// SIMATIC STEP 7 (V5.x) project CP#01_OB_PLC(TATA)
// CPU: CPU 315-2 DP
// station: P_ADR_BUS
// station: Hardware
// station: OB_PLC_PC-11
// program: S7 Program(1)

SYMBOL_TABLE
"CMD TO BEC"	DB 10	DB 10	// Command To BEC
"FB FROMBEC"	DB 11	DB 11	// Feedback From BEC
"HMI TAGS"	DB 35	DB 35	// HMI Tags are here
"RDREC"	SFB 52	SFB 52	// Read a Process Data Record
"WRREC"	SFB 53	SFB 53	// Write a Process Data Record
"RD_SINFO"	SFC 6	SFC 6	// Read OB Start Information
"BLKMOV"	SFC 20	SFC 20	// Copy Variables
"FILL"	SFC 21	SFC 21	// Initialize a Memory Area
"RDSYSST"	SFC 51	SFC 51	// Read a System Status List or Partial List
"WR_REC"	SFC 58	SFC 58	// Write Data Record
"RD_REC"	SFC 59	SFC 59	// Read a Data Record
END_SYMBOL_TABLE

// FB 7: know-how protected block, not included

// FB 8: know-how protected block, not included

FUNCTION_BLOCK FB 102
VERSION : 0.0
BEGIN
// body was compiled from an SCL source; compiled code not shown
END_FUNCTION_BLOCK

FUNCTION_BLOCK FB 103
VERSION : 0.0
BEGIN
// body was compiled from an SCL source; compiled code not shown
END_FUNCTION_BLOCK

FUNCTION_BLOCK FB 108
VERSION : 0.0
BEGIN
// body was compiled from an SCL source; compiled code not shown
END_FUNCTION_BLOCK

FUNCTION_BLOCK FB 109
VERSION : 0.0
BEGIN
// body was compiled from an SCL source; compiled code not shown
END_FUNCTION_BLOCK

// FC 1: know-how protected block, not included

// FC 2: know-how protected block, not included

// FC 3: know-how protected block, not included

// FC 4: know-how protected block, not included

FUNCTION FC 10 : VOID
AUTHOR : SKD
NAME : CDSPL
VERSION : 0.1
BEGIN
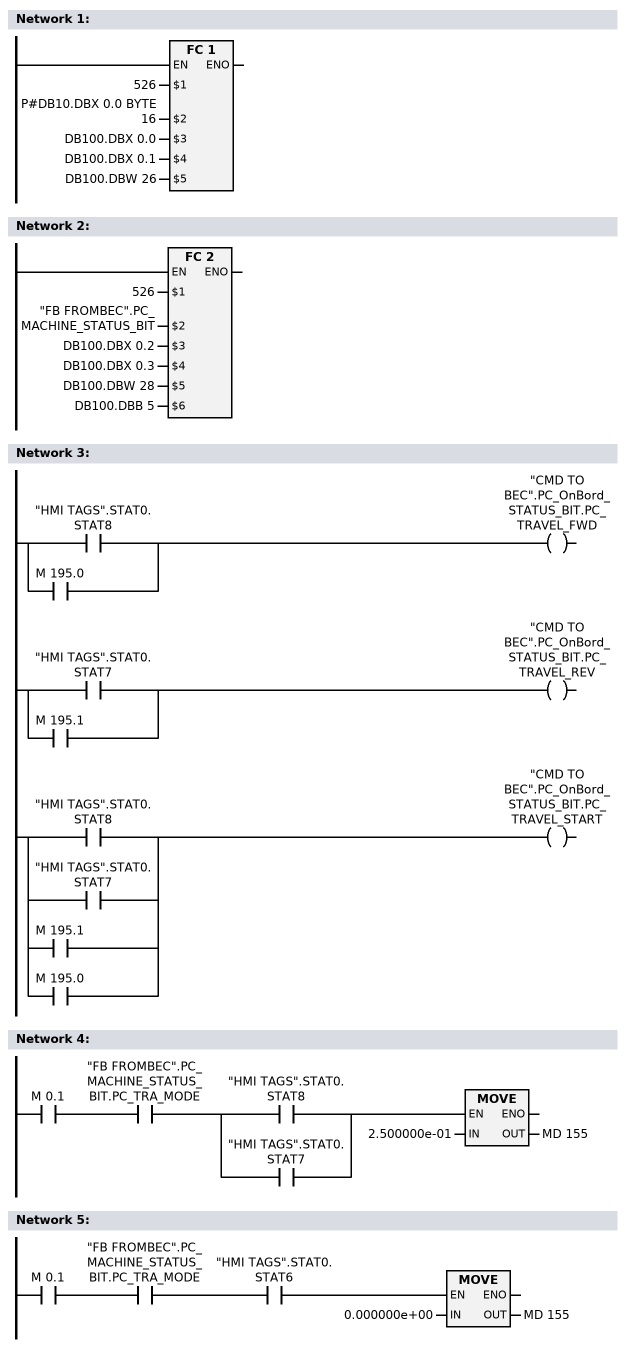
NETWORK
TITLE =
      CALL  FC 1 (
           $1                       := 526,
           $2                       := P#DB10.DBX 0.0 BYTE 16,
           $3                       := DB100.DBX 0.0,
           $4                       := DB100.DBX 0.1,
           $5                       := DB100.DBW 26);
      NOP   0;
NETWORK
TITLE =
      CALL  FC 2 (
           $1                       := 526,
           $2                       := "FB FROMBEC".PC_MACHINE_STATUS_BIT,
           $3                       := DB100.DBX 0.2,
           $4                       := DB100.DBX 0.3,
           $5                       := DB100.DBW 28,
           $6                       := DB100.DBB 5);
      NOP   0;
NETWORK
TITLE =
      O     "HMI TAGS".STAT0.STAT8;
      O     M 195.0;
      =     "CMD TO BEC".PC_OnBord_STATUS_BIT.PC_TRAVEL_FWD;
      O     "HMI TAGS".STAT0.STAT7;
      O     M 195.1;
      =     "CMD TO BEC".PC_OnBord_STATUS_BIT.PC_TRAVEL_REV;
      O     "HMI TAGS".STAT0.STAT8;
      O     "HMI TAGS".STAT0.STAT7;
      O     M 195.1;
      O     M 195.0;
      =     "CMD TO BEC".PC_OnBord_STATUS_BIT.PC_TRAVEL_START;
NETWORK
TITLE =
      A     M 0.1;
      A     "FB FROMBEC".PC_MACHINE_STATUS_BIT.PC_TRA_MODE;
      A(;
      O     "HMI TAGS".STAT0.STAT8;
      O     "HMI TAGS".STAT0.STAT7;
      );
      JNB   _001;
      L     2.500000e-01;
      T     MD 155;
_001: NOP   0;
NETWORK
TITLE =
      A     M 0.1;
      A     "FB FROMBEC".PC_MACHINE_STATUS_BIT.PC_TRA_MODE;
      A     "HMI TAGS".STAT0.STAT6;
      JNB   _002;
      L     0.000000e+00;
      T     MD 155;
_002: NOP   0;
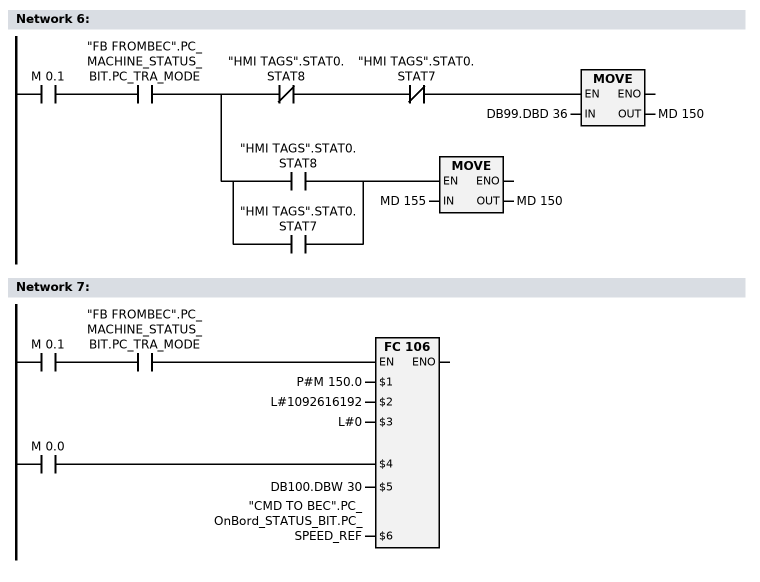
NETWORK
TITLE =
      A     M 0.1;
      A     "FB FROMBEC".PC_MACHINE_STATUS_BIT.PC_TRA_MODE;
      =     L 0.0;
      A     L 0.0;
      AN    "HMI TAGS".STAT0.STAT8;
      AN    "HMI TAGS".STAT0.STAT7;
      JNB   _003;
      L     DB99.DBD 36;
      T     MD 150;
_003: NOP   0;
      A     L 0.0;
      A(;
      O     "HMI TAGS".STAT0.STAT8;
      O     "HMI TAGS".STAT0.STAT7;
      );
      JNB   _004;
      L     MD 155;
      T     MD 150;
_004: NOP   0;
NETWORK
TITLE =
      A     M 0.0;
      =     L 0.0;
      BLD   103;
      A     M 0.1;
      A     "FB FROMBEC".PC_MACHINE_STATUS_BIT.PC_TRA_MODE;
      JNB   _005;
      CALL  FC 106 (
           $1                       := P#M 150.0,
           $2                       := L#1092616192,
           $3                       := L#0,
           $4                       := L 0.0,
           $5                       := DB100.DBW 30,
           $6                       := "CMD TO BEC".PC_OnBord_STATUS_BIT.PC_SPEED_REF);
_005: NOP   0;
END_FUNCTION

FUNCTION FC 14 : VOID
VERSION : 0.1
BEGIN
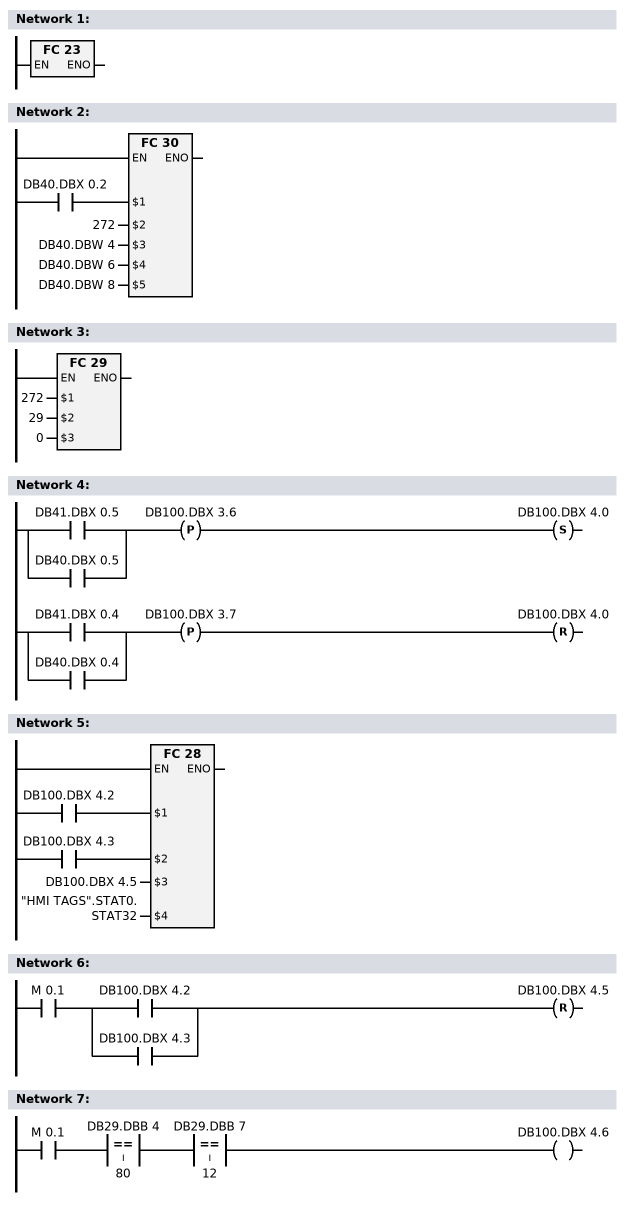
NETWORK
TITLE =
      CALL  FC 23;
      NOP   0;
NETWORK
TITLE =
      A     DB40.DBX 0.2;
      =     L 0.0;
      BLD   103;
      CALL  FC 30 (
           $1                       := L 0.0,
           $2                       := 272,
           $3                       := DB40.DBW 4,
           $4                       := DB40.DBW 6,
           $5                       := DB40.DBW 8);
      NOP   0;
NETWORK
TITLE =
      CALL  FC 29 (
           $1                       := 272,
           $2                       := 29,
           $3                       := 0);
      NOP   0;
NETWORK
TITLE =
      A(;
      O     DB41.DBX 0.5;
      O     DB40.DBX 0.5;
      );
      FP    DB100.DBX 3.6;
      S     DB100.DBX 4.0;
      A(;
      O     DB41.DBX 0.4;
      O     DB40.DBX 0.4;
      );
      FP    DB100.DBX 3.7;
      R     DB100.DBX 4.0;
      NOP   0;
NETWORK
TITLE =
      A     DB100.DBX 4.2;
      =     L 0.0;
      BLD   103;
      A     DB100.DBX 4.3;
      =     L 0.1;
      BLD   103;
      CALL  FC 28 (
           $1                       := L 0.0,
           $2                       := L 0.1,
           $3                       := DB100.DBX 4.5,
           $4                       := "HMI TAGS".STAT0.STAT32);
      NOP   0;
NETWORK
TITLE =
      A     M 0.1;
      A(;
      O     DB100.DBX 4.2;
      O     DB100.DBX 4.3;
      );
      R     DB100.DBX 4.5;
NETWORK
TITLE =
      A     M 0.1;
      A(;
      L     DB29.DBB 4;
      L     80;
      ==I;
      );
      A(;
      L     DB29.DBB 7;
      L     12;
      ==I;
      );
      =     DB100.DBX 4.6;
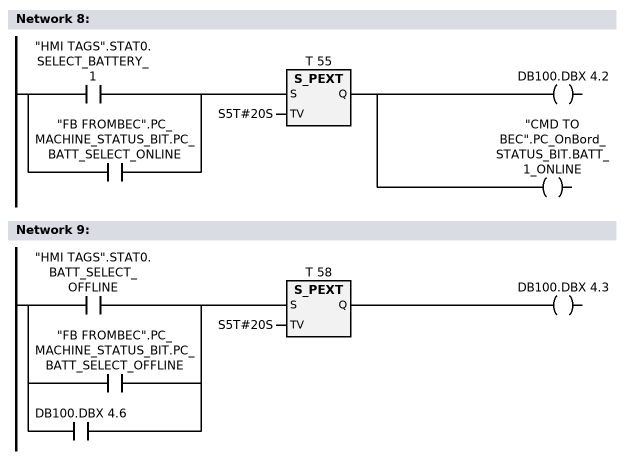
NETWORK
TITLE =
      A(;
      O     "HMI TAGS".STAT0.SELECT_BATTERY_1;
      O     "FB FROMBEC".PC_MACHINE_STATUS_BIT.PC_BATT_SELECT_ONLINE;
      );
      L     S5T#20S;
      SE    T 55;
      NOP   0;
      NOP   0;
      NOP   0;
      A     T 55;
      =     DB100.DBX 4.2;
      =     "CMD TO BEC".PC_OnBord_STATUS_BIT.BATT_1_ONLINE;
NETWORK
TITLE =
      A(;
      O     "HMI TAGS".STAT0.BATT_SELECT_OFFLINE;
      O     "FB FROMBEC".PC_MACHINE_STATUS_BIT.PC_BATT_SELECT_OFFLINE;
      O     DB100.DBX 4.6;
      );
      L     S5T#20S;
      SE    T 58;
      NOP   0;
      NOP   0;
      NOP   0;
      A     T 58;
      =     DB100.DBX 4.3;
END_FUNCTION

FUNCTION FC 16 : VOID
VERSION : 0.1
BEGIN
// (block stored without names or comments; labels and parameter names are numbered)
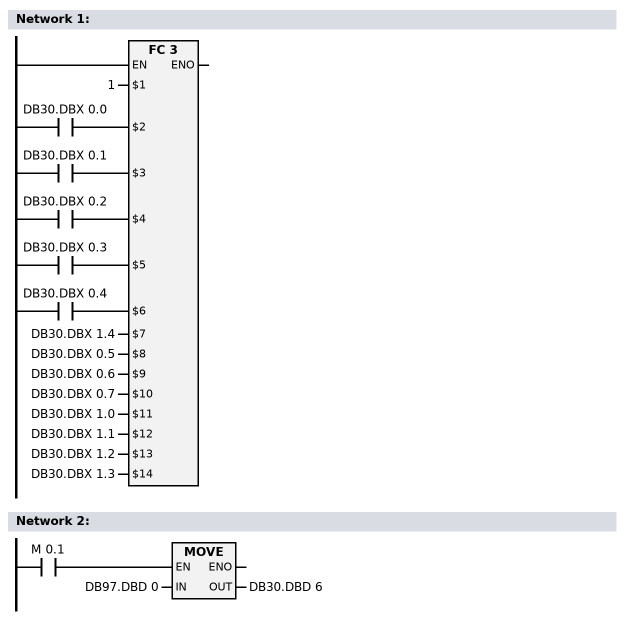
NETWORK
TITLE =
      A     DB30.DBX 0.0;
      =     L 4.0;
      BLD   103;
      A     DB30.DBX 0.1;
      =     L 4.1;
      BLD   103;
      A     DB30.DBX 0.2;
      =     L 4.2;
      BLD   103;
      A     DB30.DBX 0.3;
      =     L 4.3;
      BLD   103;
      A     DB30.DBX 0.4;
      =     L 4.4;
      BLD   103;
      CALL  FC 3 (
           $1                       := 1,
           $2                       := L 4.0,
           $3                       := L 4.1,
           $4                       := L 4.2,
           $5                       := L 4.3,
           $6                       := L 4.4,
           $7                       := DB30.DBX 1.4,
           $8                       := DB30.DBX 0.5,
           $9                       := DB30.DBX 0.6,
           $10                      := DB30.DBX 0.7,
           $11                      := DB30.DBX 1.0,
           $12                      := DB30.DBX 1.1,
           $13                      := DB30.DBX 1.2,
           $14                      := DB30.DBX 1.3);
      NOP   0;
NETWORK
TITLE =
      A     M 0.1;
      JNB   M001;
      L     DB97.DBD 0;
      T     DB30.DBD 6;
M001: NOP   0;
END_FUNCTION

FUNCTION FC 19 : VOID
VERSION : 0.1
BEGIN
// (block stored without names or comments; labels and parameter names are numbered)
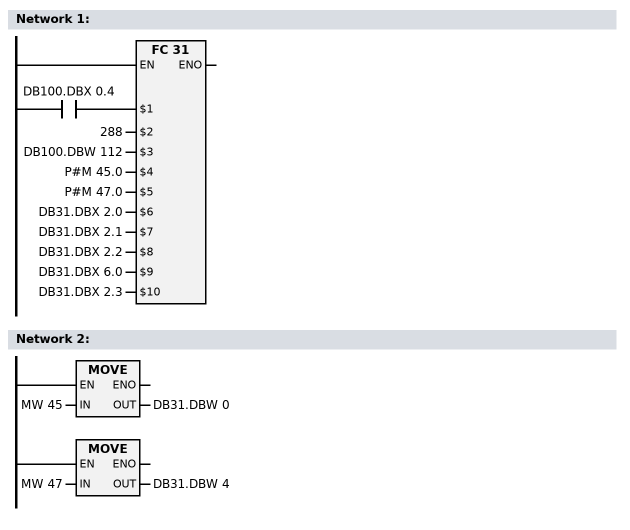
NETWORK
TITLE =
      A     DB100.DBX 0.4;
      =     L 0.0;
      BLD   103;
      CALL  FC 31 (
           $1                       := L 0.0,
           $2                       := 288,
           $3                       := DB100.DBW 112,
           $4                       := P#M 45.0,
           $5                       := P#M 47.0,
           $6                       := DB31.DBX 2.0,
           $7                       := DB31.DBX 2.1,
           $8                       := DB31.DBX 2.2,
           $9                       := DB31.DBX 6.0,
           $10                      := DB31.DBX 2.3);
      NOP   0;
NETWORK
TITLE =
      L     MW 45;
      T     DB31.DBW 0;
      L     MW 47;
      T     DB31.DBW 4;
END_FUNCTION

FUNCTION FC 20 : VOID
VERSION : 0.1
BEGIN
// (block stored without names or comments; labels and parameter names are numbered)
NETWORK
TITLE =
      A     M 0.1;
      A(;
      L     DB21.DBW 46;
      L     1;
      ==I;
      );
      A(;
      L     DB21.DBB 50;
      L     'P';
      ==I;
      );
      JNB   M001;
      L     DB21.DBW 24;
      T     "HMI TAGS".STAT98.STAT120;
M001: NOP   0;
NETWORK
TITLE =
      A     M 0.1;
      A(;
      L     DB21.DBW 46;
      L     1;
      ==I;
      );
      A(;
      L     DB21.DBB 50;
      L     'C';
      ==I;
      );
      A(;
      L     DB21.DBW 74;
      L     2;
      ==I;
      );
      A(;
      L     DB21.DBB 78;
      L     'P';
      ==I;
      );
      JNB   M002;
      L     DB21.DBW 52;
      T     "HMI TAGS".STAT98.STAT120;
M002: NOP   0;
NETWORK
TITLE =
      A     M 0.1;
      A(;
      L     DB21.DBW 46;
      L     1;
      ==I;
      );
      A(;
      L     DB21.DBB 50;
      L     'C';
      ==I;
      );
      A(;
      L     DB21.DBW 74;
      L     2;
      ==I;
      );
      A(;
      L     DB21.DBB 78;
      L     'C';
      ==I;
      );
      A(;
      L     DB21.DBW 102;
      L     3;
      ==I;
      );
      A(;
      L     DB21.DBB 106;
      L     'P';
      ==I;
      );
      JNB   M003;
      L     DB21.DBW 80;
      T     "HMI TAGS".STAT98.STAT120;
M003: NOP   0;
NETWORK
TITLE =
      A     M 0.1;
      A(;
      L     DB21.DBW 46;
      L     1;
      ==I;
      );
      A(;
      L     DB21.DBB 50;
      L     'C';
      ==I;
      );
      A(;
      L     DB21.DBW 74;
      L     2;
      ==I;
      );
      A(;
      L     DB21.DBB 78;
      L     'C';
      ==I;
      );
      A(;
      L     DB21.DBW 102;
      L     3;
      ==I;
      );
      A(;
      L     DB21.DBB 106;
      L     'C';
      ==I;
      );
      A(;
      L     DB21.DBW 130;
      L     4;
      ==I;
      );
      A(;
      L     DB21.DBB 134;
      L     'P';
      ==I;
      );
      JNB   M004;
      L     DB21.DBW 108;
      T     "HMI TAGS".STAT98.STAT120;
M004: NOP   0;
NETWORK
TITLE =
      A     M 0.1;
      A(;
      L     DB21.DBW 46;
      L     1;
      ==I;
      );
      A(;
      L     DB21.DBB 50;
      L     'C';
      ==I;
      );
      =     L 0.0;
      A     L 0.0;
      JNB   M005;
      L     DB21.DBW 24;
      T     "HMI TAGS".STAT98.STAT121;
M005: NOP   0;
      A     L 0.0;
      JNB   M006;
      L     DB21.DBB 50;
      T     DB35.DBB 284;
M006: NOP   0;
END_FUNCTION

FUNCTION FC 21 : VOID
VERSION : 0.1
BEGIN
// (block stored without names or comments; labels and parameter names are numbered)
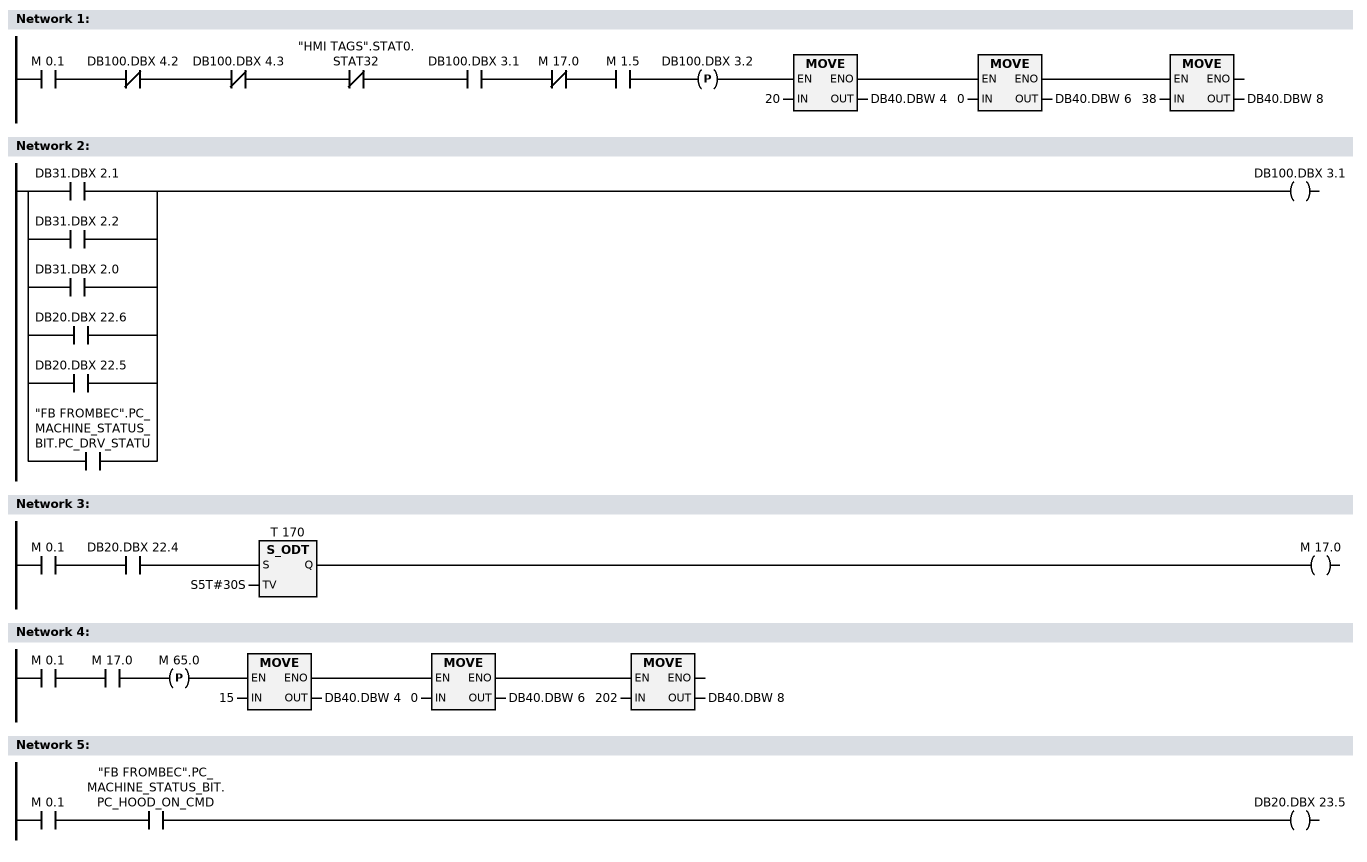
NETWORK
TITLE =
      A(;
      A(;
      A     M 0.1;
      AN    DB100.DBX 4.2;
      AN    DB100.DBX 4.3;
      AN    "HMI TAGS".STAT0.STAT32;
      A     DB100.DBX 3.1;
      AN    M 17.0;
      A     M 1.5;
      FP    DB100.DBX 3.2;
      JNB   M001;
      L     20;
      T     DB40.DBW 4;
      SET;
      SAVE;
      CLR;
M001: A     BR;
      );
      JNB   M002;
      L     0;
      T     DB40.DBW 6;
      SET;
      SAVE;
      CLR;
M002: A     BR;
      );
      JNB   M003;
      L     38;
      T     DB40.DBW 8;
M003: NOP   0;
NETWORK
TITLE =
      O     DB31.DBX 2.1;
      O     DB31.DBX 2.2;
      O     DB31.DBX 2.0;
      O     DB20.DBX 22.6;
      O     DB20.DBX 22.5;
      O     "FB FROMBEC".PC_MACHINE_STATUS_BIT.PC_DRV_STATU;
      =     DB100.DBX 3.1;
NETWORK
TITLE =
      A     M 0.1;
      A     DB20.DBX 22.4;
      L     S5T#30S;
      SD    T 170;
      NOP   0;
      NOP   0;
      NOP   0;
      A     T 170;
      =     M 17.0;
NETWORK
TITLE =
      A(;
      A(;
      A     M 0.1;
      A     M 17.0;
      FP    M 65.0;
      JNB   M004;
      L     15;
      T     DB40.DBW 4;
      SET;
      SAVE;
      CLR;
M004: A     BR;
      );
      JNB   M005;
      L     0;
      T     DB40.DBW 6;
      SET;
      SAVE;
      CLR;
M005: A     BR;
      );
      JNB   M006;
      L     202;
      T     DB40.DBW 8;
M006: NOP   0;
NETWORK
TITLE =
      A     M 0.1;
      A     "FB FROMBEC".PC_MACHINE_STATUS_BIT.PC_HOOD_ON_CMD;
      =     DB20.DBX 23.5;
NETWORK
TITLE =
      BE;
END_FUNCTION

FUNCTION FC 22 : VOID
VERSION : 0.1
BEGIN
// (block stored without names or comments; labels and parameter names are numbered)
NETWORK
TITLE =
      A     DB41.DBX 0.4;
      A(;
      L     DB29.DBB 8;
      L     B#16#3;
      ==I;
      );
      A(;
      L     DB29.DBB 11;
      L     32;
      ==I;
      );
      =     DB100.DBX 15.1;
      A     DB100.DBX 15.1;
      JNB   M001;
      CALL  "FILL" (
           BVAL                     := P#DB29.DBX 0.0 BYTE 30,
           RET_VAL                  := DB100.DBW 122,
           BLK                      := P#DB17.DBX 0.0 BYTE 30);
M001: NOP   0;
NETWORK
TITLE =
      A     DB41.DBX 0.4;
      A(;
      L     DB29.DBB 8;
      L     B#16#4;
      ==I;
      );
      A(;
      L     DB29.DBB 11;
      L     30;
      ==I;
      );
      =     DB100.DBX 15.2;
      A     DB100.DBX 15.2;
      JNB   M002;
      CALL  "FILL" (
           BVAL                     := P#DB29.DBX 0.0 BYTE 30,
           RET_VAL                  := DB100.DBW 124,
           BLK                      := P#DB19.DBX 0.0 BYTE 30);
M002: NOP   0;
NETWORK
TITLE =
      A     DB41.DBX 0.4;
      A(;
      L     DB29.DBB 8;
      L     B#16#5;
      ==I;
      );
      A(;
      L     DB29.DBB 11;
      L     34;
      ==I;
      );
      =     DB100.DBX 15.3;
      A     DB100.DBX 15.3;
      FP    DB100.DBX 15.5;
      JNB   M003;
      CALL  "FILL" (
           BVAL                     := P#DB29.DBX 0.0 BYTE 34,
           RET_VAL                  := DB100.DBW 126,
           BLK                      := P#DB18.DBX 0.0 BYTE 34);
M003: NOP   0;
NETWORK
TITLE =
      A     DB41.DBX 0.4;
      A(;
      L     DB29.DBB 8;
      L     B#16#10;
      ==I;
      );
      A(;
      L     DB29.DBB 11;
      L     167;
      ==I;
      );
      =     DB100.DBX 15.4;
      A     DB100.DBX 15.4;
      JNB   M004;
      CALL  "FILL" (
           BVAL                     := P#DB29.DBX 0.0 BYTE 167,
           RET_VAL                  := DB100.DBW 128,
           BLK                      := P#DB21.DBX 0.0 BYTE 167);
M004: NOP   0;
END_FUNCTION

FUNCTION FC 23 : VOID
VERSION : 0.1
BEGIN
// (block stored without names or comments; labels and parameter names are numbered)
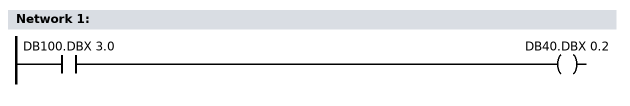
NETWORK
TITLE =
      A     DB100.DBX 3.0;
      =     DB40.DBX 0.2;
END_FUNCTION

FUNCTION FC 24 : VOID
VERSION : 0.1
BEGIN
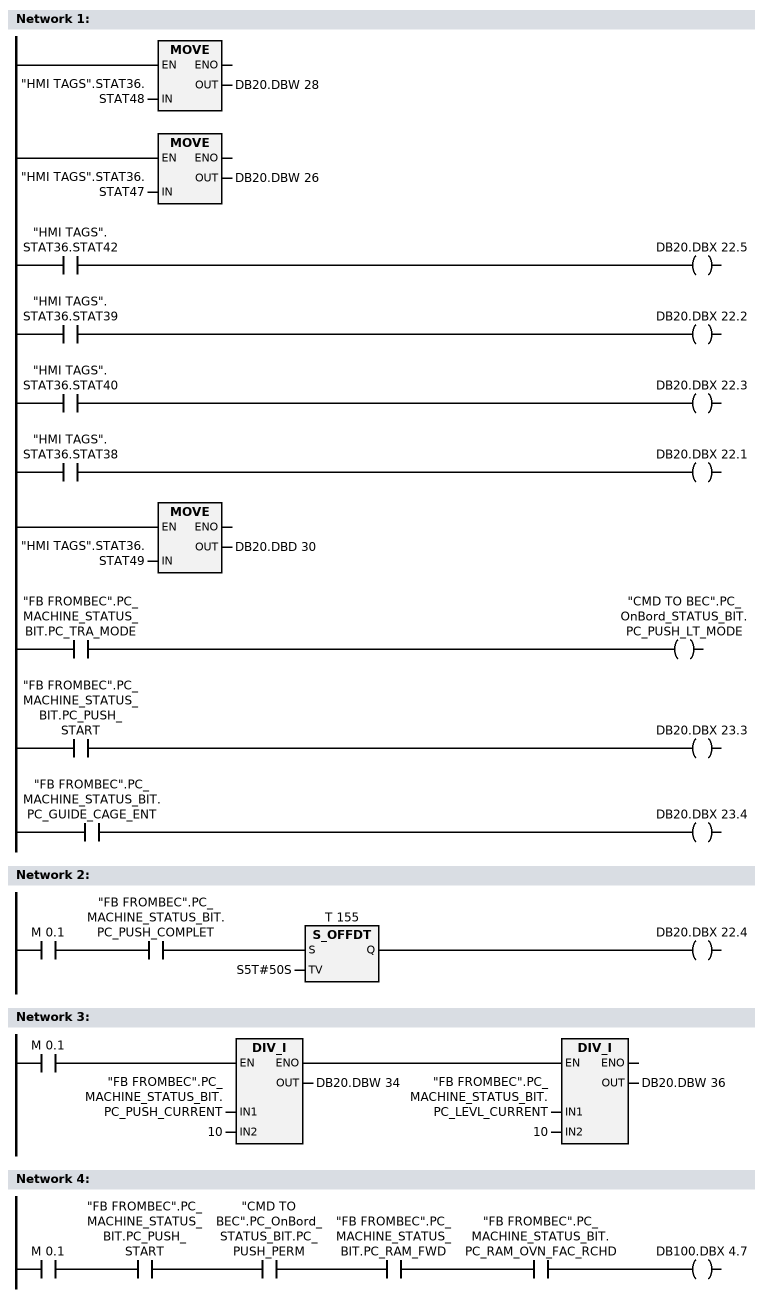
NETWORK
TITLE =
      L     "HMI TAGS".STAT36.STAT48;
      T     DB20.DBW 28;
      L     "HMI TAGS".STAT36.STAT47;
      T     DB20.DBW 26;
      A     "HMI TAGS".STAT36.STAT42;
      =     DB20.DBX 22.5;
      A     "HMI TAGS".STAT36.STAT39;
      =     DB20.DBX 22.2;
      A     "HMI TAGS".STAT36.STAT40;
      =     DB20.DBX 22.3;
      A     "HMI TAGS".STAT36.STAT38;
      =     DB20.DBX 22.1;
      L     "HMI TAGS".STAT36.STAT49;
      T     DB20.DBD 30;
      A     "FB FROMBEC".PC_MACHINE_STATUS_BIT.PC_TRA_MODE;
      =     "CMD TO BEC".PC_OnBord_STATUS_BIT.PC_PUSH_LT_MODE;
      A     "FB FROMBEC".PC_MACHINE_STATUS_BIT.PC_PUSH_START;
      =     DB20.DBX 23.3;
      A     "FB FROMBEC".PC_MACHINE_STATUS_BIT.PC_GUIDE_CAGE_ENT;
      =     DB20.DBX 23.4;
NETWORK
TITLE =
      A     M 0.1;
      A     "FB FROMBEC".PC_MACHINE_STATUS_BIT.PC_PUSH_COMPLET;
      L     S5T#50S;
      SF    T 155;
      NOP   0;
      NOP   0;
      NOP   0;
      A     T 155;
      =     DB20.DBX 22.4;
NETWORK
TITLE =
      A(;
      A     M 0.1;
      JNB   _001;
      L     "FB FROMBEC".PC_MACHINE_STATUS_BIT.PC_PUSH_CURRENT;
      L     10;
      /I;
      T     DB20.DBW 34;
      AN    OV;
      SAVE;
      CLR;
_001: A     BR;
      );
      JNB   _002;
      L     "FB FROMBEC".PC_MACHINE_STATUS_BIT.PC_LEVL_CURRENT;
      L     10;
      /I;
      T     DB20.DBW 36;
_002: NOP   0;
NETWORK
TITLE =
      A     M 0.1;
      A     "FB FROMBEC".PC_MACHINE_STATUS_BIT.PC_PUSH_START;
      A     "CMD TO BEC".PC_OnBord_STATUS_BIT.PC_PUSH_PERM;
      A     "FB FROMBEC".PC_MACHINE_STATUS_BIT.PC_RAM_FWD;
      A     "FB FROMBEC".PC_MACHINE_STATUS_BIT.PC_RAM_OVN_FAC_RCHD;
      =     DB100.DBX 4.7;
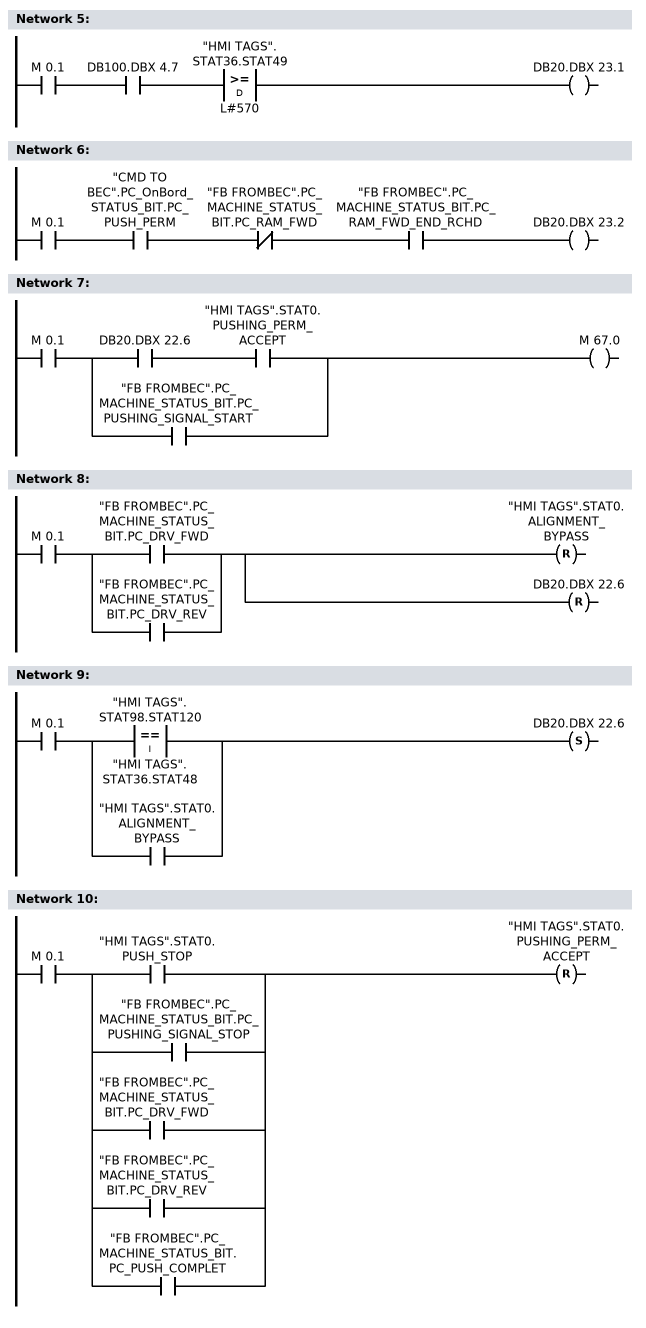
NETWORK
TITLE =
      A     M 0.1;
      A     DB100.DBX 4.7;
      A(;
      L     "HMI TAGS".STAT36.STAT49;
      L     L#570;
      >=D;
      );
      =     DB20.DBX 23.1;
NETWORK
TITLE =
      A     M 0.1;
      A     "CMD TO BEC".PC_OnBord_STATUS_BIT.PC_PUSH_PERM;
      AN    "FB FROMBEC".PC_MACHINE_STATUS_BIT.PC_RAM_FWD;
      A     "FB FROMBEC".PC_MACHINE_STATUS_BIT.PC_RAM_FWD_END_RCHD;
      =     DB20.DBX 23.2;
NETWORK
TITLE =
      A     M 0.1;
      A(;
      A     DB20.DBX 22.6;
      A     "HMI TAGS".STAT0.PUSHING_PERM_ACCEPT;
      O     "FB FROMBEC".PC_MACHINE_STATUS_BIT.PC_PUSHING_SIGNAL_START;
      );
      =     M 67.0;
NETWORK
TITLE =
      A     M 0.1;
      A(;
      O     "FB FROMBEC".PC_MACHINE_STATUS_BIT.PC_DRV_FWD;
      O     "FB FROMBEC".PC_MACHINE_STATUS_BIT.PC_DRV_REV;
      );
      R     "HMI TAGS".STAT0.ALIGNMENT_BYPASS;
      R     DB20.DBX 22.6;
NETWORK
TITLE =
      A     M 0.1;
      A(;
      O(;
      L     "HMI TAGS".STAT98.STAT120;
      L     "HMI TAGS".STAT36.STAT48;
      ==I;
      );
      O     "HMI TAGS".STAT0.ALIGNMENT_BYPASS;
      );
      S     DB20.DBX 22.6;
NETWORK
TITLE =
      A     M 0.1;
      A(;
      O     "HMI TAGS".STAT0.PUSH_STOP;
      O     "FB FROMBEC".PC_MACHINE_STATUS_BIT.PC_PUSHING_SIGNAL_STOP;
      O     "FB FROMBEC".PC_MACHINE_STATUS_BIT.PC_DRV_FWD;
      O     "FB FROMBEC".PC_MACHINE_STATUS_BIT.PC_DRV_REV;
      O     "FB FROMBEC".PC_MACHINE_STATUS_BIT.PC_PUSH_COMPLET;
      );
      R     "HMI TAGS".STAT0.PUSHING_PERM_ACCEPT;
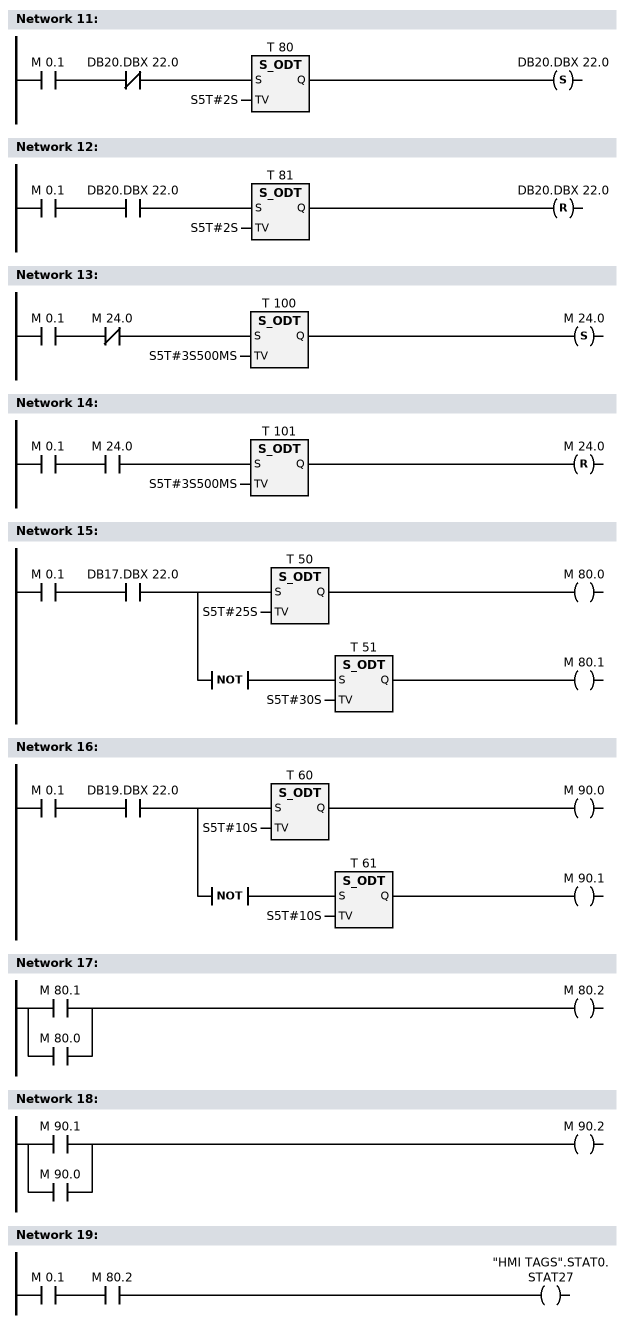
NETWORK
TITLE =
      A     M 0.1;
      AN    DB20.DBX 22.0;
      L     S5T#2S;
      SD    T 80;
      NOP   0;
      NOP   0;
      NOP   0;
      A     T 80;
      S     DB20.DBX 22.0;
NETWORK
TITLE =
      A     M 0.1;
      A     DB20.DBX 22.0;
      L     S5T#2S;
      SD    T 81;
      NOP   0;
      NOP   0;
      NOP   0;
      A     T 81;
      R     DB20.DBX 22.0;
NETWORK
TITLE =
      A     M 0.1;
      AN    M 24.0;
      L     S5T#3S500MS;
      SD    T 100;
      NOP   0;
      NOP   0;
      NOP   0;
      A     T 100;
      S     M 24.0;
NETWORK
TITLE =
      A     M 0.1;
      A     M 24.0;
      L     S5T#3S500MS;
      SD    T 101;
      NOP   0;
      NOP   0;
      NOP   0;
      A     T 101;
      R     M 24.0;
NETWORK
TITLE =
      A     M 0.1;
      A     DB17.DBX 22.0;
      =     L 0.0;
      A     L 0.0;
      L     S5T#25S;
      SD    T 50;
      NOP   0;
      NOP   0;
      NOP   0;
      A     T 50;
      =     M 80.0;
      A     L 0.0;
      NOT;
      L     S5T#30S;
      SD    T 51;
      NOP   0;
      NOP   0;
      NOP   0;
      A     T 51;
      =     M 80.1;
NETWORK
TITLE =
      A     M 0.1;
      A     DB19.DBX 22.0;
      =     L 0.0;
      A     L 0.0;
      L     S5T#10S;
      SD    T 60;
      NOP   0;
      NOP   0;
      NOP   0;
      A     T 60;
      =     M 90.0;
      A     L 0.0;
      NOT;
      L     S5T#10S;
      SD    T 61;
      NOP   0;
      NOP   0;
      NOP   0;
      A     T 61;
      =     M 90.1;
NETWORK
TITLE =
      O     M 80.1;
      O     M 80.0;
      =     M 80.2;
NETWORK
TITLE =
      O     M 90.1;
      O     M 90.0;
      =     M 90.2;
NETWORK
TITLE =
      A     M 0.1;
      A     M 80.2;
      =     "HMI TAGS".STAT0.STAT27;
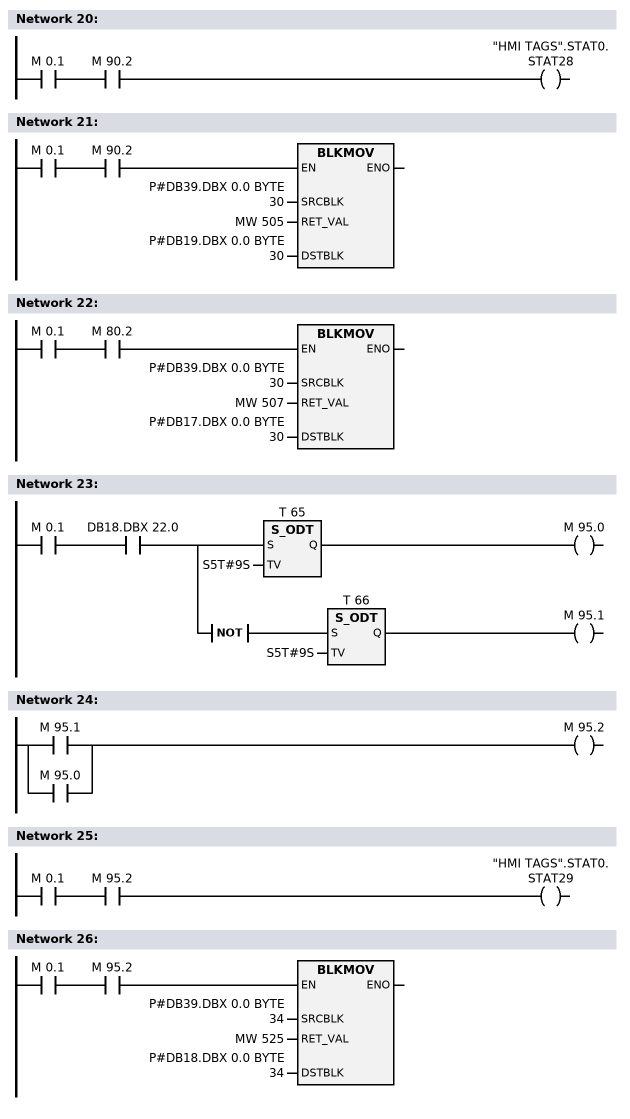
NETWORK
TITLE =
      A     M 0.1;
      A     M 90.2;
      =     "HMI TAGS".STAT0.STAT28;
NETWORK
TITLE =
      A     M 0.1;
      A     M 90.2;
      JNB   _003;
      CALL  "BLKMOV" (
           SRCBLK                   := P#DB39.DBX 0.0 BYTE 30,
           RET_VAL                  := MW 505,
           DSTBLK                   := P#DB19.DBX 0.0 BYTE 30);
_003: NOP   0;
NETWORK
TITLE =
      A     M 0.1;
      A     M 80.2;
      JNB   _004;
      CALL  "BLKMOV" (
           SRCBLK                   := P#DB39.DBX 0.0 BYTE 30,
           RET_VAL                  := MW 507,
           DSTBLK                   := P#DB17.DBX 0.0 BYTE 30);
_004: NOP   0;
NETWORK
TITLE =
      A     M 0.1;
      A     DB18.DBX 22.0;
      =     L 0.0;
      A     L 0.0;
      L     S5T#9S;
      SD    T 65;
      NOP   0;
      NOP   0;
      NOP   0;
      A     T 65;
      =     M 95.0;
      A     L 0.0;
      NOT;
      L     S5T#9S;
      SD    T 66;
      NOP   0;
      NOP   0;
      NOP   0;
      A     T 66;
      =     M 95.1;
NETWORK
TITLE =
      O     M 95.1;
      O     M 95.0;
      =     M 95.2;
NETWORK
TITLE =
      A     M 0.1;
      A     M 95.2;
      =     "HMI TAGS".STAT0.STAT29;
NETWORK
TITLE =
      A     M 0.1;
      A     M 95.2;
      JNB   _005;
      CALL  "BLKMOV" (
           SRCBLK                   := P#DB39.DBX 0.0 BYTE 34,
           RET_VAL                  := MW 525,
           DSTBLK                   := P#DB18.DBX 0.0 BYTE 34);
_005: NOP   0;
END_FUNCTION

FUNCTION FC 26 : VOID
VERSION : 0.1
BEGIN
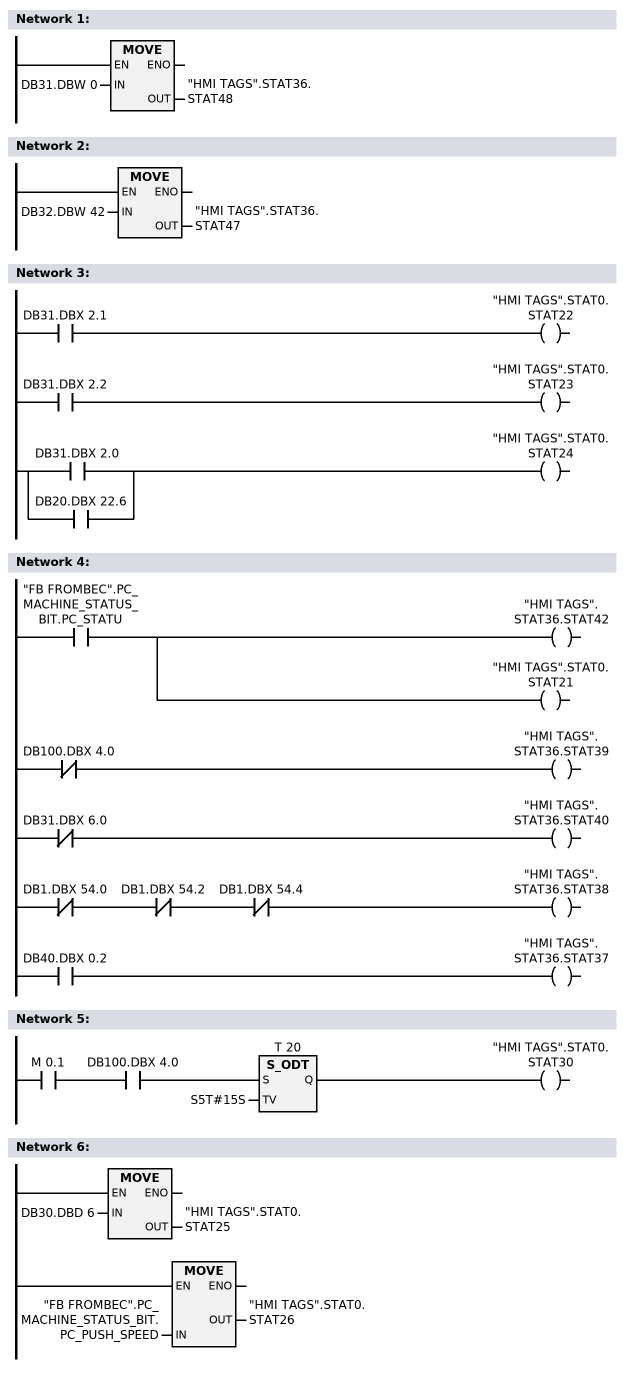
NETWORK
TITLE =
      L     DB31.DBW 0;
      T     "HMI TAGS".STAT36.STAT48;
NETWORK
TITLE =
      L     DB32.DBW 42;
      T     "HMI TAGS".STAT36.STAT47;
NETWORK
TITLE =
      A     DB31.DBX 2.1;
      =     "HMI TAGS".STAT0.STAT22;
      A     DB31.DBX 2.2;
      =     "HMI TAGS".STAT0.STAT23;
      O     DB31.DBX 2.0;
      O     DB20.DBX 22.6;
      =     "HMI TAGS".STAT0.STAT24;
NETWORK
TITLE =
      A     "FB FROMBEC".PC_MACHINE_STATUS_BIT.PC_STATU;
      =     "HMI TAGS".STAT36.STAT42;
      =     "HMI TAGS".STAT0.STAT21;
      AN    DB100.DBX 4.0;
      =     "HMI TAGS".STAT36.STAT39;
      AN    DB31.DBX 6.0;
      =     "HMI TAGS".STAT36.STAT40;
      AN    DB1.DBX 54.0;
      AN    DB1.DBX 54.2;
      AN    DB1.DBX 54.4;
      =     "HMI TAGS".STAT36.STAT38;
      A     DB40.DBX 0.2;
      =     "HMI TAGS".STAT36.STAT37;
NETWORK
TITLE =
      A     M 0.1;
      A     DB100.DBX 4.0;
      L     S5T#15S;
      SD    T 20;
      NOP   0;
      NOP   0;
      NOP   0;
      A     T 20;
      =     "HMI TAGS".STAT0.STAT30;
NETWORK
TITLE =
      L     DB30.DBD 6;
      T     "HMI TAGS".STAT0.STAT25;
      L     "FB FROMBEC".PC_MACHINE_STATUS_BIT.PC_PUSH_SPEED;
      T     "HMI TAGS".STAT0.STAT26;
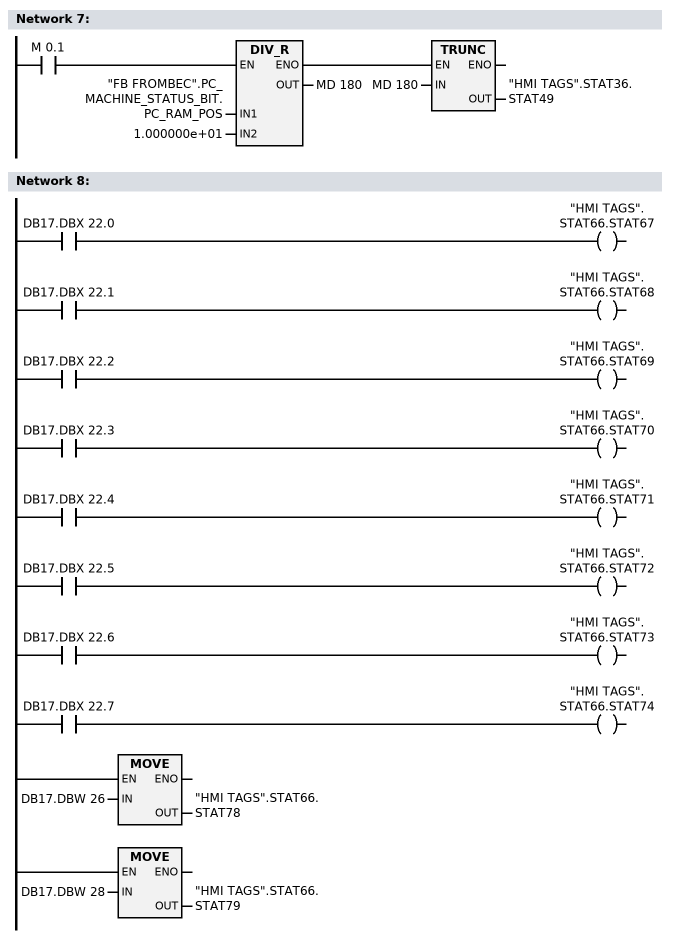
NETWORK
TITLE =
      A(;
      A     M 0.1;
      JNB   _001;
      L     "FB FROMBEC".PC_MACHINE_STATUS_BIT.PC_RAM_POS;
      L     1.000000e+01;
      /R;
      T     MD 180;
      AN    OV;
      SAVE;
      CLR;
_001: A     BR;
      );
      JNB   _002;
      L     MD 180;
      TRUNC;
      T     "HMI TAGS".STAT36.STAT49;
_002: NOP   0;
NETWORK
TITLE =
      A     DB17.DBX 22.0;
      =     "HMI TAGS".STAT66.STAT67;
      A     DB17.DBX 22.1;
      =     "HMI TAGS".STAT66.STAT68;
      A     DB17.DBX 22.2;
      =     "HMI TAGS".STAT66.STAT69;
      A     DB17.DBX 22.3;
      =     "HMI TAGS".STAT66.STAT70;
      A     DB17.DBX 22.4;
      =     "HMI TAGS".STAT66.STAT71;
      A     DB17.DBX 22.5;
      =     "HMI TAGS".STAT66.STAT72;
      A     DB17.DBX 22.6;
      =     "HMI TAGS".STAT66.STAT73;
      A     DB17.DBX 22.7;
      =     "HMI TAGS".STAT66.STAT74;
      L     DB17.DBW 26;
      T     "HMI TAGS".STAT66.STAT78;
      L     DB17.DBW 28;
      T     "HMI TAGS".STAT66.STAT79;
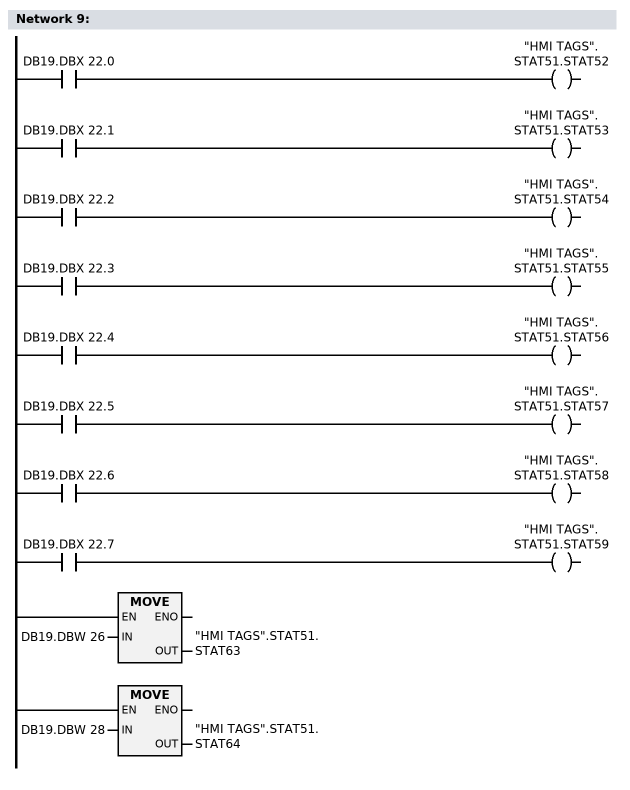
NETWORK
TITLE =
      A     DB19.DBX 22.0;
      =     "HMI TAGS".STAT51.STAT52;
      A     DB19.DBX 22.1;
      =     "HMI TAGS".STAT51.STAT53;
      A     DB19.DBX 22.2;
      =     "HMI TAGS".STAT51.STAT54;
      A     DB19.DBX 22.3;
      =     "HMI TAGS".STAT51.STAT55;
      A     DB19.DBX 22.4;
      =     "HMI TAGS".STAT51.STAT56;
      A     DB19.DBX 22.5;
      =     "HMI TAGS".STAT51.STAT57;
      A     DB19.DBX 22.6;
      =     "HMI TAGS".STAT51.STAT58;
      A     DB19.DBX 22.7;
      =     "HMI TAGS".STAT51.STAT59;
      L     DB19.DBW 26;
      T     "HMI TAGS".STAT51.STAT63;
      L     DB19.DBW 28;
      T     "HMI TAGS".STAT51.STAT64;
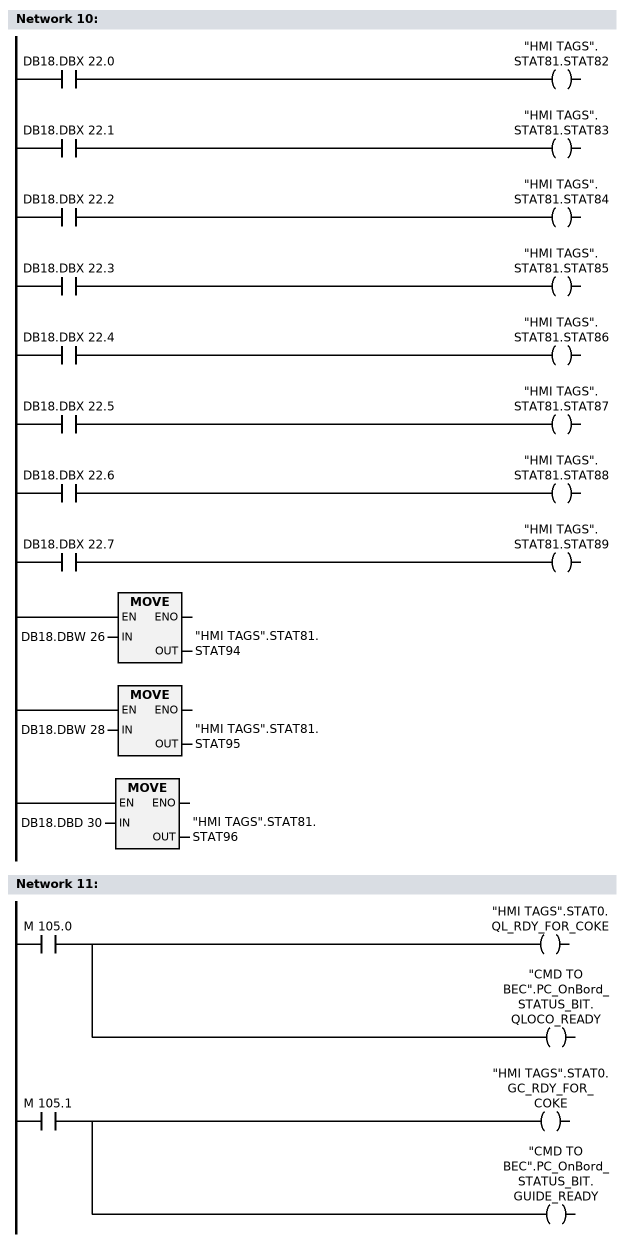
NETWORK
TITLE =
      A     DB18.DBX 22.0;
      =     "HMI TAGS".STAT81.STAT82;
      A     DB18.DBX 22.1;
      =     "HMI TAGS".STAT81.STAT83;
      A     DB18.DBX 22.2;
      =     "HMI TAGS".STAT81.STAT84;
      A     DB18.DBX 22.3;
      =     "HMI TAGS".STAT81.STAT85;
      A     DB18.DBX 22.4;
      =     "HMI TAGS".STAT81.STAT86;
      A     DB18.DBX 22.5;
      =     "HMI TAGS".STAT81.STAT87;
      A     DB18.DBX 22.6;
      =     "HMI TAGS".STAT81.STAT88;
      A     DB18.DBX 22.7;
      =     "HMI TAGS".STAT81.STAT89;
      L     DB18.DBW 26;
      T     "HMI TAGS".STAT81.STAT94;
      L     DB18.DBW 28;
      T     "HMI TAGS".STAT81.STAT95;
      L     DB18.DBD 30;
      T     "HMI TAGS".STAT81.STAT96;
NETWORK
TITLE =
      A     M 105.0;
      =     "HMI TAGS".STAT0.QL_RDY_FOR_COKE;
      =     "CMD TO BEC".PC_OnBord_STATUS_BIT.QLOCO_READY;
      A     M 105.1;
      =     "HMI TAGS".STAT0.GC_RDY_FOR_COKE;
      =     "CMD TO BEC".PC_OnBord_STATUS_BIT.GUIDE_READY;
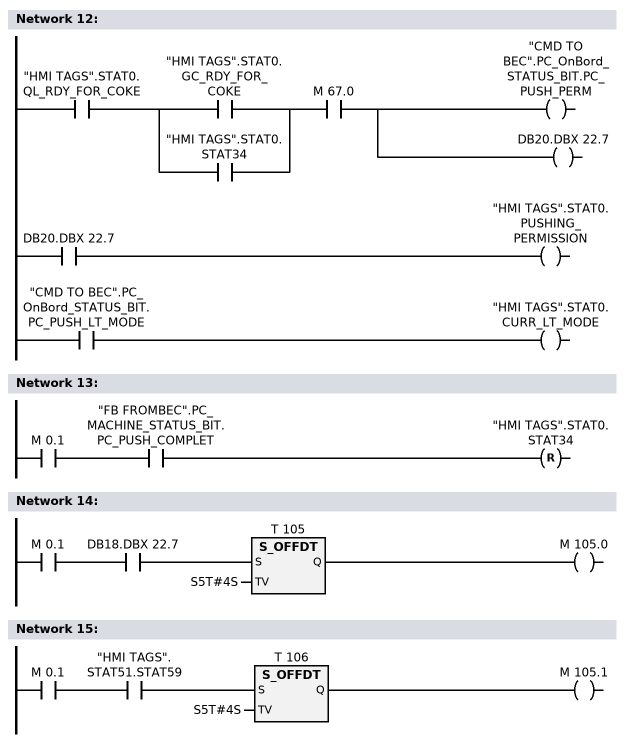
NETWORK
TITLE =
      A     "HMI TAGS".STAT0.QL_RDY_FOR_COKE;
      A(;
      O     "HMI TAGS".STAT0.GC_RDY_FOR_COKE;
      O     "HMI TAGS".STAT0.STAT34;
      );
      A     M 67.0;
      =     "CMD TO BEC".PC_OnBord_STATUS_BIT.PC_PUSH_PERM;
      =     DB20.DBX 22.7;
      A     DB20.DBX 22.7;
      =     "HMI TAGS".STAT0.PUSHING_PERMISSION;
      A     "CMD TO BEC".PC_OnBord_STATUS_BIT.PC_PUSH_LT_MODE;
      =     "HMI TAGS".STAT0.CURR_LT_MODE;
NETWORK
TITLE =
      A     M 0.1;
      A     "FB FROMBEC".PC_MACHINE_STATUS_BIT.PC_PUSH_COMPLET;
      R     "HMI TAGS".STAT0.STAT34;
NETWORK
TITLE =
      A     M 0.1;
      A     DB18.DBX 22.7;
      L     S5T#4S;
      SF    T 105;
      NOP   0;
      NOP   0;
      NOP   0;
      A     T 105;
      =     M 105.0;
NETWORK
TITLE =
      A     M 0.1;
      A     "HMI TAGS".STAT51.STAT59;
      L     S5T#4S;
      SF    T 106;
      NOP   0;
      NOP   0;
      NOP   0;
      A     T 106;
      =     M 105.1;
END_FUNCTION

FUNCTION FC 27 : VOID
VERSION : 0.1
BEGIN
// (block stored without names or comments; labels and parameter names are numbered)
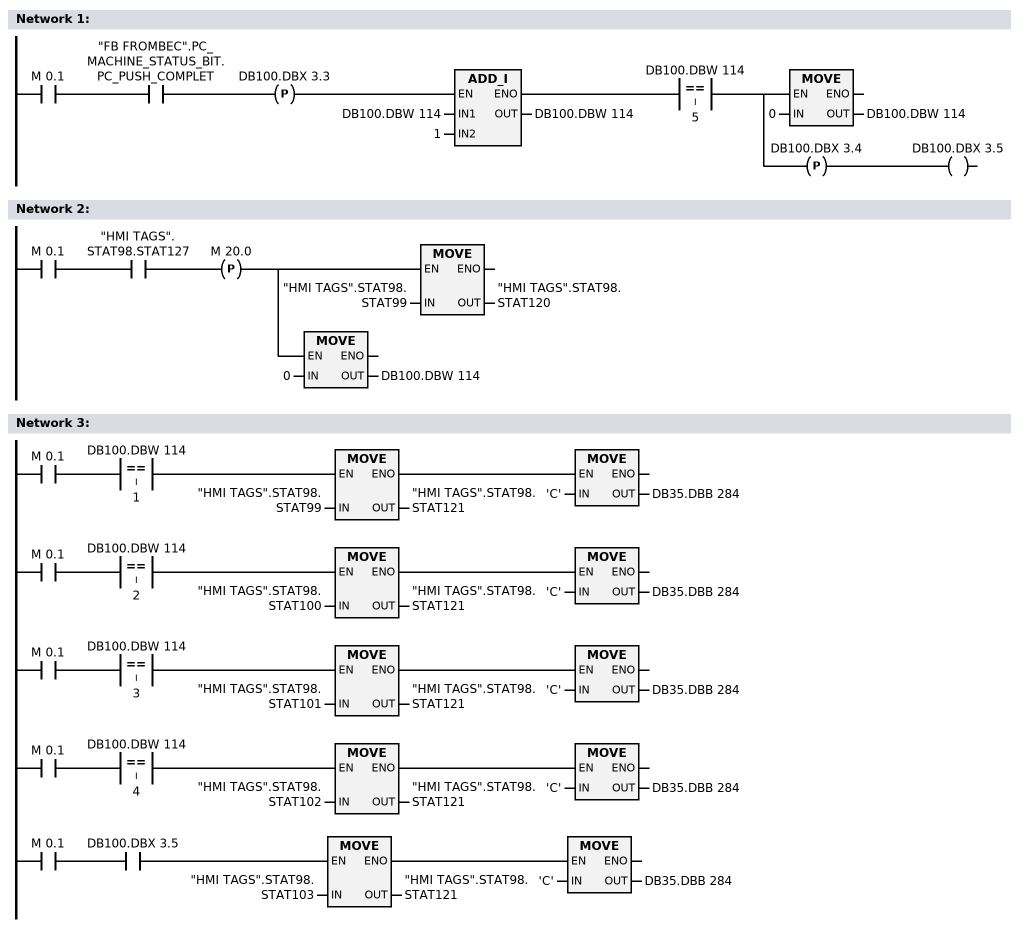
NETWORK
TITLE =
      A(;
      A     M 0.1;
      A     "FB FROMBEC".PC_MACHINE_STATUS_BIT.PC_PUSH_COMPLET;
      FP    DB100.DBX 3.3;
      JNB   M001;
      L     DB100.DBW 114;
      L     1;
      +I;
      T     DB100.DBW 114;
      AN    OV;
      SAVE;
      CLR;
M001: A     BR;
      );
      A(;
      L     DB100.DBW 114;
      L     5;
      ==I;
      );
      =     L 0.0;
      A     L 0.0;
      JNB   M002;
      L     0;
      T     DB100.DBW 114;
M002: NOP   0;
      A     L 0.0;
      FP    DB100.DBX 3.4;
      =     DB100.DBX 3.5;
NETWORK
TITLE =
      A     M 0.1;
      A     "HMI TAGS".STAT98.STAT127;
      FP    M 20.0;
      =     L 0.0;
      A     L 0.0;
      JNB   M003;
      L     "HMI TAGS".STAT98.STAT99;
      T     "HMI TAGS".STAT98.STAT120;
M003: NOP   0;
      A     L 0.0;
      JNB   M004;
      L     0;
      T     DB100.DBW 114;
M004: NOP   0;
NETWORK
TITLE =
      A     M 0.1;
      =     L 0.0;
      A(;
      A     L 0.0;
      A(;
      L     DB100.DBW 114;
      L     1;
      ==I;
      );
      JNB   M005;
      L     "HMI TAGS".STAT98.STAT99;
      T     "HMI TAGS".STAT98.STAT121;
      SET;
      SAVE;
      CLR;
M005: A     BR;
      );
      JNB   M006;
      L     'C';
      T     DB35.DBB 284;
M006: NOP   0;
      A(;
      A     L 0.0;
      A(;
      L     DB100.DBW 114;
      L     2;
      ==I;
      );
      JNB   M007;
      L     "HMI TAGS".STAT98.STAT100;
      T     "HMI TAGS".STAT98.STAT121;
      SET;
      SAVE;
      CLR;
M007: A     BR;
      );
      JNB   M008;
      L     'C';
      T     DB35.DBB 284;
M008: NOP   0;
      A(;
      A     L 0.0;
      A(;
      L     DB100.DBW 114;
      L     3;
      ==I;
      );
      JNB   M009;
      L     "HMI TAGS".STAT98.STAT101;
      T     "HMI TAGS".STAT98.STAT121;
      SET;
      SAVE;
      CLR;
M009: A     BR;
      );
      JNB   M010;
      L     'C';
      T     DB35.DBB 284;
M010: NOP   0;
      A(;
      A     L 0.0;
      A(;
      L     DB100.DBW 114;
      L     4;
      ==I;
      );
      JNB   M011;
      L     "HMI TAGS".STAT98.STAT102;
      T     "HMI TAGS".STAT98.STAT121;
      SET;
      SAVE;
      CLR;
M011: A     BR;
      );
      JNB   M012;
      L     'C';
      T     DB35.DBB 284;
M012: NOP   0;
      A(;
      A     L 0.0;
      A     DB100.DBX 3.5;
      JNB   M013;
      L     "HMI TAGS".STAT98.STAT103;
      T     "HMI TAGS".STAT98.STAT121;
      SET;
      SAVE;
      CLR;
M013: A     BR;
      );
      JNB   M014;
      L     'C';
      T     DB35.DBB 284;
M014: NOP   0;
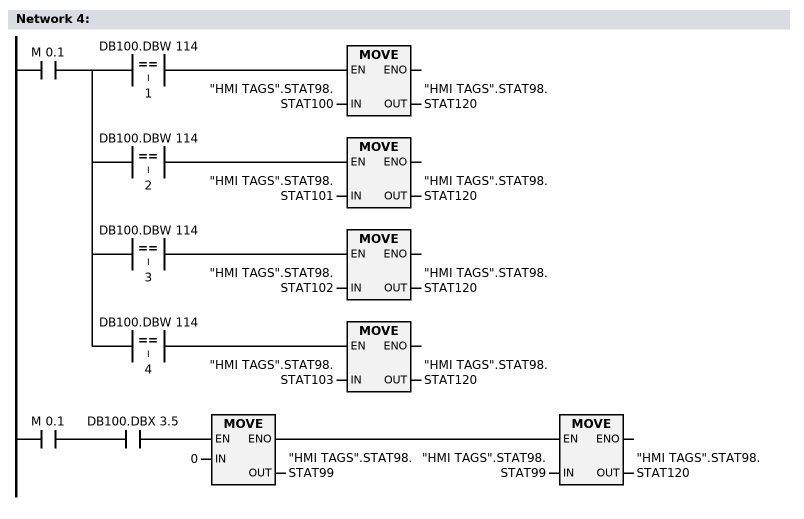
NETWORK
TITLE =
      A     M 0.1;
      =     L 0.0;
      A     L 0.0;
      A(;
      L     DB100.DBW 114;
      L     1;
      ==I;
      );
      JNB   M015;
      L     "HMI TAGS".STAT98.STAT100;
      T     "HMI TAGS".STAT98.STAT120;
M015: NOP   0;
      A     L 0.0;
      A(;
      L     DB100.DBW 114;
      L     2;
      ==I;
      );
      JNB   M016;
      L     "HMI TAGS".STAT98.STAT101;
      T     "HMI TAGS".STAT98.STAT120;
M016: NOP   0;
      A     L 0.0;
      A(;
      L     DB100.DBW 114;
      L     3;
      ==I;
      );
      JNB   M017;
      L     "HMI TAGS".STAT98.STAT102;
      T     "HMI TAGS".STAT98.STAT120;
M017: NOP   0;
      A     L 0.0;
      A(;
      L     DB100.DBW 114;
      L     4;
      ==I;
      );
      JNB   M018;
      L     "HMI TAGS".STAT98.STAT103;
      T     "HMI TAGS".STAT98.STAT120;
M018: NOP   0;
      A(;
      A     L 0.0;
      A     DB100.DBX 3.5;
      JNB   M019;
      L     0;
      T     "HMI TAGS".STAT98.STAT99;
      SET;
      SAVE;
      CLR;
M019: A     BR;
      );
      JNB   M020;
      L     "HMI TAGS".STAT98.STAT99;
      T     "HMI TAGS".STAT98.STAT120;
M020: NOP   0;
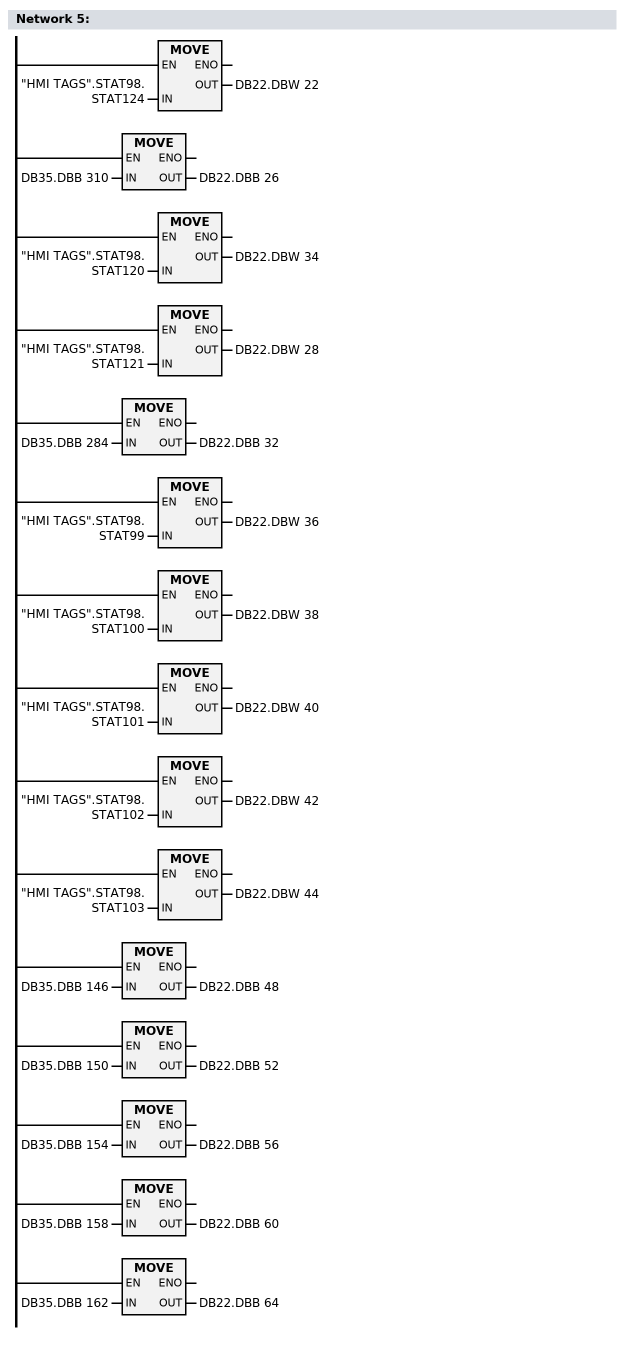
NETWORK
TITLE =
      L     "HMI TAGS".STAT98.STAT124;
      T     DB22.DBW 22;
      L     DB35.DBB 310;
      T     DB22.DBB 26;
      L     "HMI TAGS".STAT98.STAT120;
      T     DB22.DBW 34;
      L     "HMI TAGS".STAT98.STAT121;
      T     DB22.DBW 28;
      L     DB35.DBB 284;
      T     DB22.DBB 32;
      L     "HMI TAGS".STAT98.STAT99;
      T     DB22.DBW 36;
      L     "HMI TAGS".STAT98.STAT100;
      T     DB22.DBW 38;
      L     "HMI TAGS".STAT98.STAT101;
      T     DB22.DBW 40;
      L     "HMI TAGS".STAT98.STAT102;
      T     DB22.DBW 42;
      L     "HMI TAGS".STAT98.STAT103;
      T     DB22.DBW 44;
      L     DB35.DBB 146;
      T     DB22.DBB 48;
      L     DB35.DBB 150;
      T     DB22.DBB 52;
      L     DB35.DBB 154;
      T     DB22.DBB 56;
      L     DB35.DBB 158;
      T     DB22.DBB 60;
      L     DB35.DBB 162;
      T     DB22.DBB 64;
END_FUNCTION

FUNCTION FC 28 : VOID
VERSION : 0.1
BEGIN
// (block stored without names or comments; labels and parameter names are numbered)
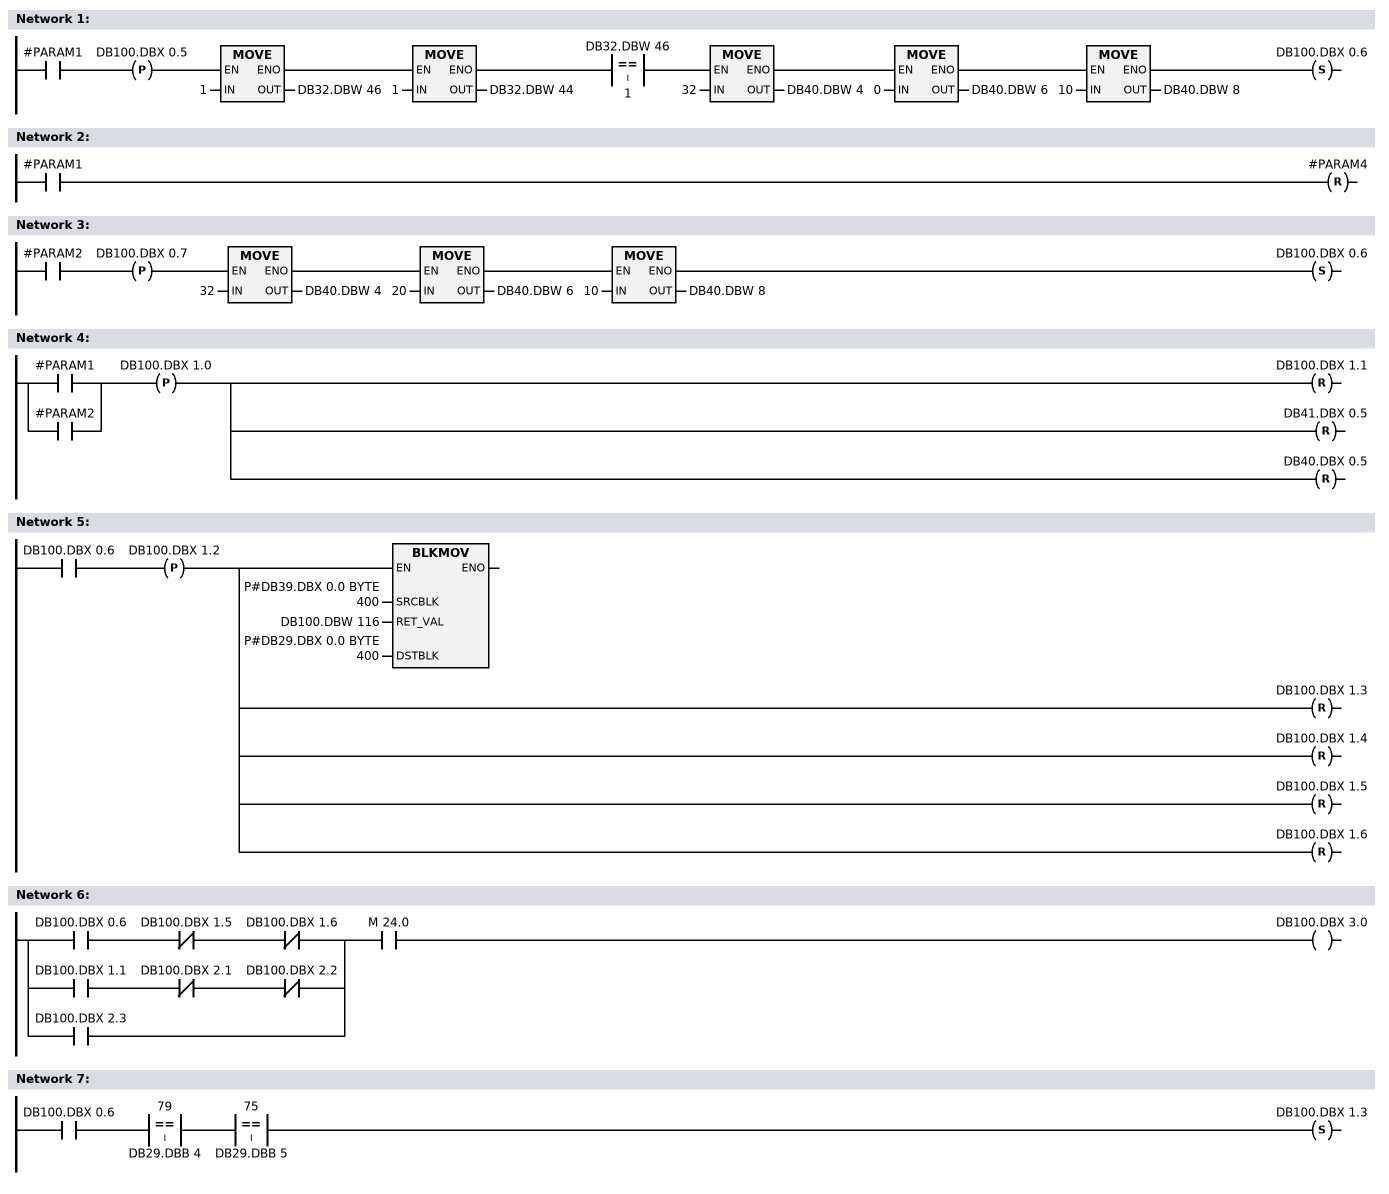
NETWORK
TITLE =
      A(;
      A(;
      A(;
      A(;
      A     #PARAM1;
      FP    DB100.DBX 0.5;
      JNB   M001;
      L     1;
      T     DB32.DBW 46;
      SET;
      SAVE;
      CLR;
M001: A     BR;
      );
      JNB   M002;
      L     1;
      T     DB32.DBW 44;
      SET;
      SAVE;
      CLR;
M002: A     BR;
      );
      A(;
      L     DB32.DBW 46;
      L     1;
      ==I;
      );
      JNB   M003;
      L     32;
      T     DB40.DBW 4;
      SET;
      SAVE;
      CLR;
M003: A     BR;
      );
      JNB   M004;
      L     0;
      T     DB40.DBW 6;
      SET;
      SAVE;
      CLR;
M004: A     BR;
      );
      JNB   M005;
      L     10;
      T     DB40.DBW 8;
      SET;
      SAVE;
      CLR;
M005: A     BR;
      S     DB100.DBX 0.6;
NETWORK
TITLE =
      A     #PARAM1;
      R     #PARAM4;
NETWORK
TITLE =
      A(;
      A(;
      A     #PARAM2;
      FP    DB100.DBX 0.7;
      JNB   M006;
      L     32;
      T     DB40.DBW 4;
      SET;
      SAVE;
      CLR;
M006: A     BR;
      );
      JNB   M007;
      L     20;
      T     DB40.DBW 6;
      SET;
      SAVE;
      CLR;
M007: A     BR;
      );
      JNB   M008;
      L     10;
      T     DB40.DBW 8;
      SET;
      SAVE;
      CLR;
M008: A     BR;
      S     DB100.DBX 0.6;
NETWORK
TITLE =
      A(;
      O     #PARAM1;
      O     #PARAM2;
      );
      FP    DB100.DBX 1.0;
      R     DB100.DBX 1.1;
      R     DB41.DBX 0.5;
      R     DB40.DBX 0.5;
NETWORK
TITLE =
      A     DB100.DBX 0.6;
      FP    DB100.DBX 1.2;
      =     L 0.0;
      A     L 0.0;
      JNB   M009;
      CALL  "BLKMOV" (
           SRCBLK                   := P#DB39.DBX 0.0 BYTE 400,
           RET_VAL                  := DB100.DBW 116,
           DSTBLK                   := P#DB29.DBX 0.0 BYTE 400);
M009: NOP   0;
      A     L 0.0;
      BLD   102;
      R     DB100.DBX 1.3;
      A     L 0.0;
      BLD   102;
      R     DB100.DBX 1.4;
      A     L 0.0;
      BLD   102;
      R     DB100.DBX 1.5;
      A     L 0.0;
      BLD   102;
      R     DB100.DBX 1.6;
NETWORK
TITLE =
      A(;
      A     DB100.DBX 0.6;
      AN    DB100.DBX 1.5;
      AN    DB100.DBX 1.6;
      O;
      A     DB100.DBX 1.1;
      AN    DB100.DBX 2.1;
      AN    DB100.DBX 2.2;
      O     DB100.DBX 2.3;
      );
      A     M 24.0;
      =     DB100.DBX 3.0;
NETWORK
TITLE =
      A     DB100.DBX 0.6;
      A(;
      L     79;
      L     DB29.DBB 4;
      ==I;
      );
      A(;
      L     75;
      L     DB29.DBB 5;
      ==I;
      );
      S     DB100.DBX 1.3;
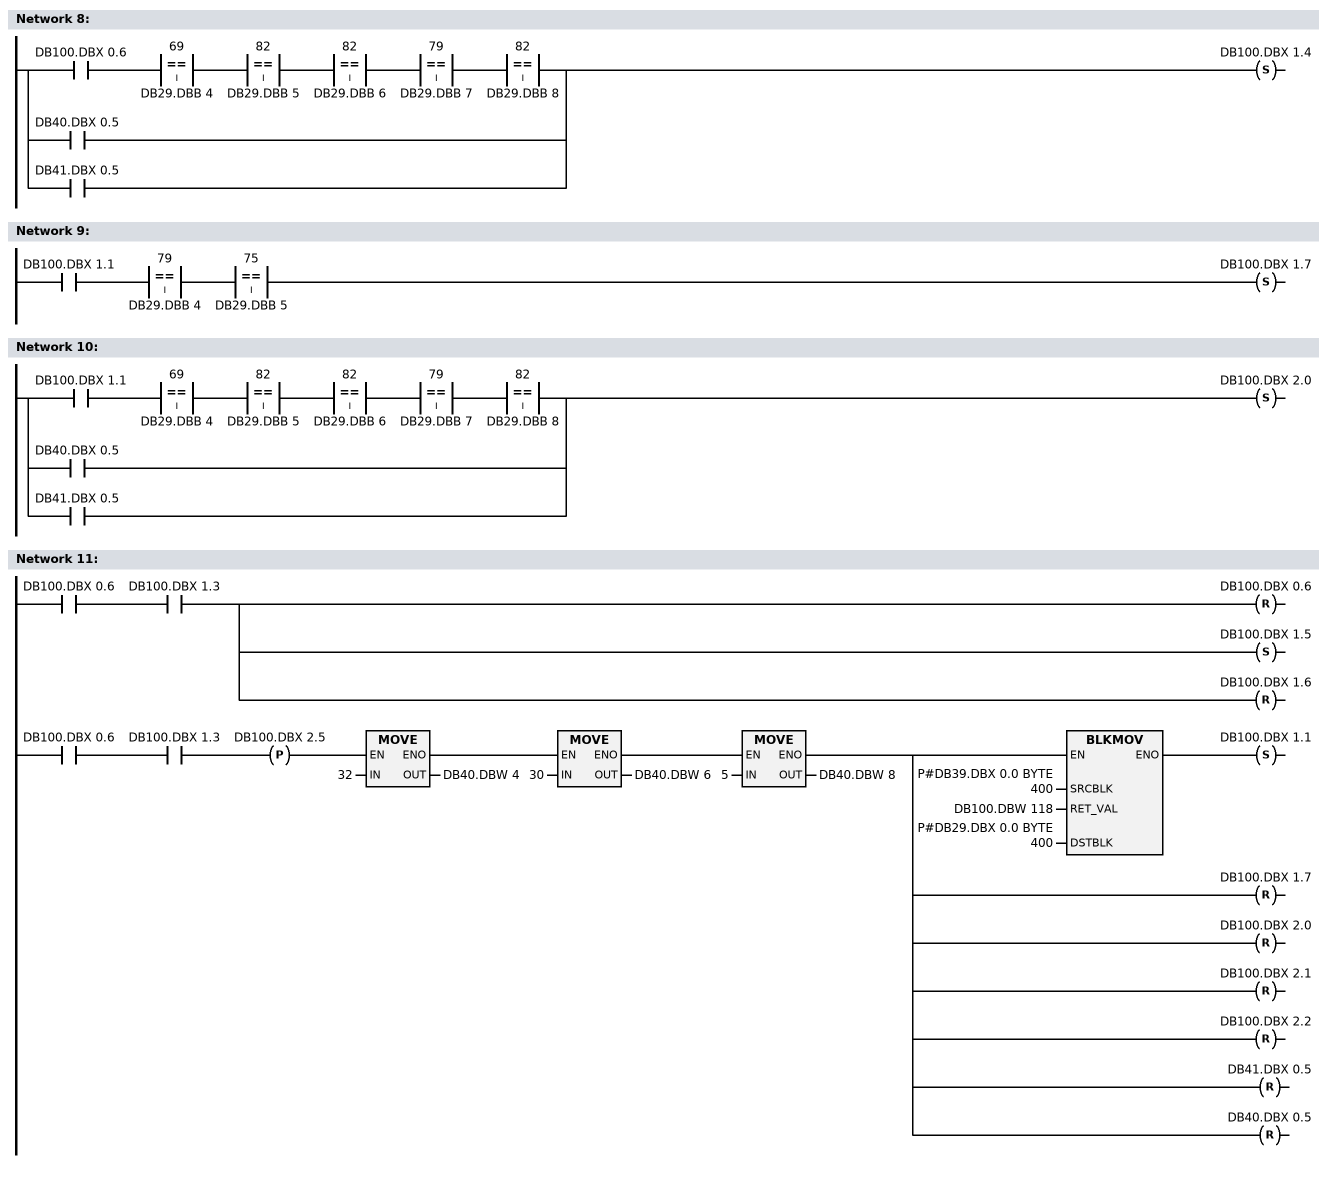
NETWORK
TITLE =
      A     DB100.DBX 0.6;
      A(;
      L     69;
      L     DB29.DBB 4;
      ==I;
      );
      A(;
      L     82;
      L     DB29.DBB 5;
      ==I;
      );
      A(;
      L     82;
      L     DB29.DBB 6;
      ==I;
      );
      A(;
      L     79;
      L     DB29.DBB 7;
      ==I;
      );
      A(;
      L     82;
      L     DB29.DBB 8;
      ==I;
      );
      O     DB40.DBX 0.5;
      O     DB41.DBX 0.5;
      S     DB100.DBX 1.4;
NETWORK
TITLE =
      A     DB100.DBX 1.1;
      A(;
      L     79;
      L     DB29.DBB 4;
      ==I;
      );
      A(;
      L     75;
      L     DB29.DBB 5;
      ==I;
      );
      S     DB100.DBX 1.7;
NETWORK
TITLE =
      A     DB100.DBX 1.1;
      A(;
      L     69;
      L     DB29.DBB 4;
      ==I;
      );
      A(;
      L     82;
      L     DB29.DBB 5;
      ==I;
      );
      A(;
      L     82;
      L     DB29.DBB 6;
      ==I;
      );
      A(;
      L     79;
      L     DB29.DBB 7;
      ==I;
      );
      A(;
      L     82;
      L     DB29.DBB 8;
      ==I;
      );
      O     DB40.DBX 0.5;
      O     DB41.DBX 0.5;
      S     DB100.DBX 2.0;
NETWORK
TITLE =
      A     DB100.DBX 0.6;
      A     DB100.DBX 1.3;
      =     L 0.0;
      A     L 0.0;
      BLD   102;
      R     DB100.DBX 0.6;
      A     L 0.0;
      BLD   102;
      S     DB100.DBX 1.5;
      A     L 0.0;
      BLD   102;
      R     DB100.DBX 1.6;
      A(;
      A(;
      A     L 0.0;
      FP    DB100.DBX 2.5;
      JNB   M010;
      L     32;
      T     DB40.DBW 4;
      SET;
      SAVE;
      CLR;
M010: A     BR;
      );
      JNB   M011;
      L     30;
      T     DB40.DBW 6;
      SET;
      SAVE;
      CLR;
M011: A     BR;
      );
      JNB   M012;
      L     5;
      T     DB40.DBW 8;
      SET;
      SAVE;
      CLR;
M012: A     BR;
      =     L 0.1;
      A     L 0.1;
      JNB   M013;
      CALL  "BLKMOV" (
           SRCBLK                   := P#DB39.DBX 0.0 BYTE 400,
           RET_VAL                  := DB100.DBW 118,
           DSTBLK                   := P#DB29.DBX 0.0 BYTE 400);
M013: A     BR;
      S     DB100.DBX 1.1;
      A     L 0.1;
      BLD   102;
      R     DB100.DBX 1.7;
      A     L 0.1;
      BLD   102;
      R     DB100.DBX 2.0;
      A     L 0.1;
      BLD   102;
      R     DB100.DBX 2.1;
      A     L 0.1;
      BLD   102;
      R     DB100.DBX 2.2;
      A     L 0.1;
      BLD   102;
      R     DB41.DBX 0.5;
      A     L 0.1;
      BLD   102;
      R     DB40.DBX 0.5;
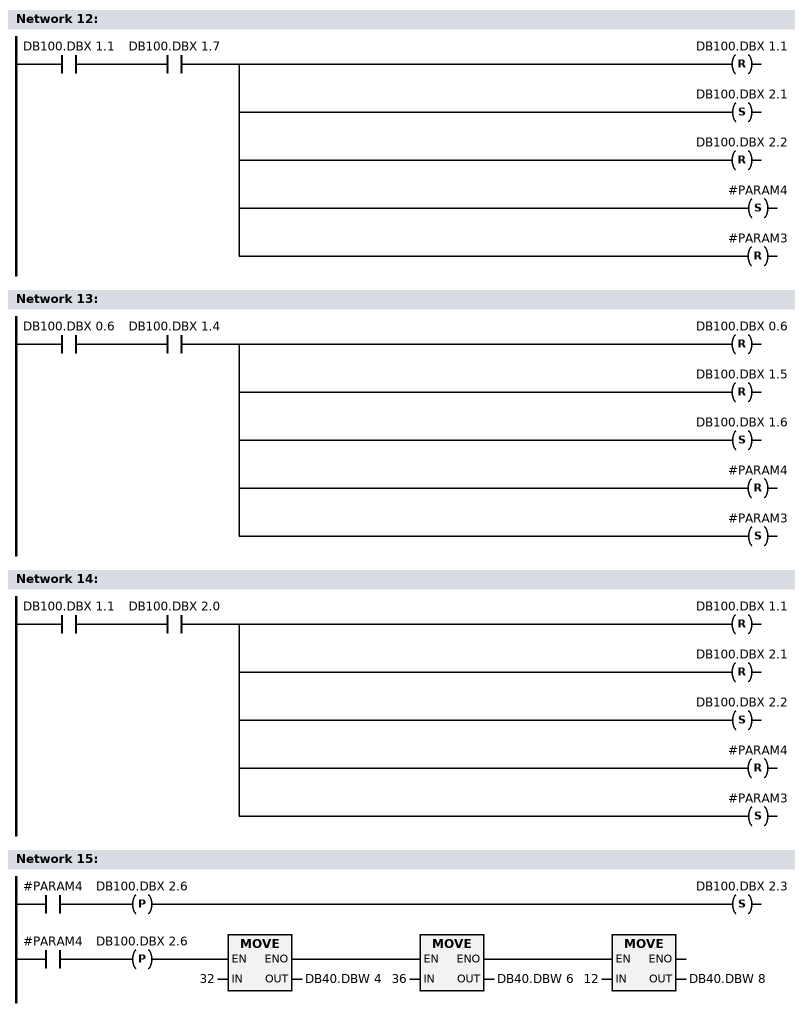
NETWORK
TITLE =
      A     DB100.DBX 1.1;
      A     DB100.DBX 1.7;
      R     DB100.DBX 1.1;
      S     DB100.DBX 2.1;
      R     DB100.DBX 2.2;
      S     #PARAM4;
      R     #PARAM3;
NETWORK
TITLE =
      A     DB100.DBX 0.6;
      A     DB100.DBX 1.4;
      R     DB100.DBX 0.6;
      R     DB100.DBX 1.5;
      S     DB100.DBX 1.6;
      R     #PARAM4;
      S     #PARAM3;
NETWORK
TITLE =
      A     DB100.DBX 1.1;
      A     DB100.DBX 2.0;
      R     DB100.DBX 1.1;
      R     DB100.DBX 2.1;
      S     DB100.DBX 2.2;
      R     #PARAM4;
      S     #PARAM3;
NETWORK
TITLE =
      A     #PARAM4;
      FP    DB100.DBX 2.6;
      =     L 0.0;
      A     L 0.0;
      BLD   102;
      S     DB100.DBX 2.3;
      A(;
      A(;
      A     L 0.0;
      JNB   M014;
      L     32;
      T     DB40.DBW 4;
      SET;
      SAVE;
      CLR;
M014: A     BR;
      );
      JNB   M015;
      L     36;
      T     DB40.DBW 6;
      SET;
      SAVE;
      CLR;
M015: A     BR;
      );
      JNB   M016;
      L     12;
      T     DB40.DBW 8;
M016: NOP   0;
NETWORK
TITLE =
NETWORK
TITLE =
NETWORK
TITLE =
      BE;
END_FUNCTION

FUNCTION FC 29 : VOID
VERSION : 0.1
BEGIN
// (block stored without names or comments; labels and parameter names are numbered)
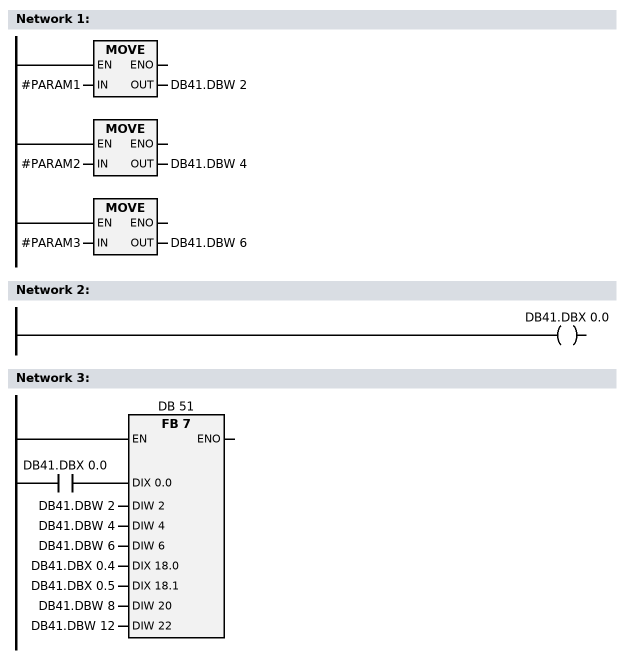
NETWORK
TITLE =
      L     #PARAM1;
      T     DB41.DBW 2;
      L     #PARAM2;
      T     DB41.DBW 4;
      L     #PARAM3;
      T     DB41.DBW 6;
NETWORK
TITLE =
      SET;
      =     DB41.DBX 0.0;
NETWORK
TITLE =
      A     DB41.DBX 0.0;
      =     L 0.0;
      BLD   103;
      CALL  FB 7 , DB 51 (
           DIX 0.0                  := L 0.0,
           DIW 2                    := DB41.DBW 2,
           DIW 4                    := DB41.DBW 4,
           DIW 6                    := DB41.DBW 6,
           DIX 18.0                 := DB41.DBX 0.4,
           DIX 18.1                 := DB41.DBX 0.5,
           DIW 20                   := DB41.DBW 8,
           DIW 22                   := DB41.DBW 12);
      NOP   0;
NETWORK
TITLE =
      AN    DB41.DBX 0.4;
      JC    M001;
      L     DB41.DBW 18;
      +     1;
      T     DB41.DBW 18;
      L     DB41.DBW 8;
      T     DB41.DBW 10;
      BE;
M001: AN    DB41.DBX 0.5;
      BEC;
      L     DB41.DBW 20;
      +     1;
      T     DB41.DBW 20;
      L     DB41.DBW 12;
      T     DB41.DBW 14;
      BE;
NETWORK
TITLE =
END_FUNCTION

FUNCTION FC 30 : VOID
VERSION : 0.1
BEGIN
// (block stored without names or comments; labels and parameter names are numbered)
